  MoveL 5993 to (239.92, 153.82, 88.06) mm, rotated rx 180 ry 0 rz -180 deg; joints [-146.88, -81.725, -27.685, 63.006, 37.821, -57.184]
  MoveL 5994 to (239.92, 153.82, 88.06) mm, rotated rx 180 ry 0 rz -180 deg; joints [-146.88, -81.725, -27.685, 63.006, 37.821, -57.184]
  Call Extruder(262.09688)
  MoveL 5995 to (239.85, 154.05, 88.06) mm, rotated rx 180 ry 0 rz 180 deg; joints [-146.86, -81.738, -27.658, 63.04, 37.832, -57.218]
  MoveL 5996 to (239.85, 154.05, 88.06) mm, rotated rx 180 ry 0 rz 180 deg; joints [-146.86, -81.738, -27.658, 63.04, 37.832, -57.218]
  Call Extruder(262.22767)
  MoveL 5997 to (239.78, 154.27, 88.06) mm, rotated rx 180 ry 0 rz -180 deg; joints [-146.84, -81.752, -27.63, 63.073, 37.842, -57.252]
  MoveL 5998 to (239.78, 154.27, 88.06) mm, rotated rx 180 ry 0 rz -180 deg; joints [-146.84, -81.752, -27.63, 63.073, 37.842, -57.252]
  Call Extruder(262.35903)
  MoveL 5999 to (239.71, 154.49, 88.06) mm, rotated rx -180 ry 0 rz 180 deg; joints [-146.82, -81.765, -27.603, 63.107, 37.853, -57.286]
  MoveL 6000 to (239.71, 154.49, 88.06) mm, rotated rx -180 ry 0 rz 180 deg; joints [-146.82, -81.765, -27.603, 63.107, 37.853, -57.286]
  Call Extruder(262.47093)
  MoveL 6001 to (239.65, 154.68, 88.06) mm, rotated rx 180 ry 0 rz 180 deg; joints [-146.803, -81.776, -27.581, 63.135, 37.862, -57.314]
  MoveL 6002 to (239.65, 154.68, 88.06) mm, rotated rx 180 ry 0 rz 180 deg; joints [-146.803, -81.776, -27.581, 63.135, 37.862, -57.314]
  Call Extruder(262.58328)
  MoveL 6003 to (239.59, 154.87, 88.06) mm, rotated rx 180 ry 0 rz 180 deg; joints [-146.785, -81.787, -27.559, 63.163, 37.872, -57.342]
  MoveL 6004 to (239.59, 154.87, 88.06) mm, rotated rx 180 ry 0 rz 180 deg; joints [-146.785, -81.787, -27.559, 63.163, 37.872, -57.342]
  Call Extruder(262.69607)
  MoveL 6005 to (239.53, 155.06, 88.06) mm, rotated rx 180 ry 0 rz 180 deg; joints [-146.768, -81.798, -27.537, 63.19, 37.881, -57.37]
  MoveL 6006 to (239.53, 155.06, 88.06) mm, rotated rx 180 ry 0 rz 180 deg; joints [-146.768, -81.798, -27.537, 63.19, 37.881, -57.37]
  Call Extruder(262.80930)
  MoveL 6007 to (239.47, 155.25, 88.06) mm, rotated rx 180 ry 0 rz 180 deg; joints [-146.751, -81.808, -27.515, 63.218, 37.891, -57.398]
  MoveL 6008 to (239.47, 155.25, 88.06) mm, rotated rx 180 ry 0 rz 180 deg; joints [-146.751, -81.808, -27.515, 63.218, 37.891, -57.398]
  Call Extruder(262.92298)
  MoveL 6009 to (239.41, 155.44, 88.06) mm, rotated rx 180 ry 0 rz 180 deg; joints [-146.734, -81.819, -27.494, 63.246, 37.9, -57.426]
  MoveL 6010 to (239.41, 155.44, 88.06) mm, rotated rx 180 ry 0 rz 180 deg; joints [-146.734, -81.819, -27.494, 63.246, 37.9, -57.426]
  Call Extruder(263.10494)
  MoveL 6011 to (239.29, 155.73, 88.06) mm, rotated rx 180 ry 0 rz -180 deg; joints [-146.706, -81.832, -27.469, 63.285, 37.918, -57.464]
  MoveL 6012 to (239.29, 155.73, 88.06) mm, rotated rx 180 ry 0 rz -180 deg; joints [-146.706, -81.832, -27.469, 63.285, 37.918, -57.464]
  Call Extruder(263.28765)
  MoveL 6013 to (239.17, 156.02, 88.06) mm, rotated rx 180 ry 0 rz -180 deg; joints [-146.678, -81.844, -27.444, 63.323, 37.936, -57.501]
  MoveL 6014 to (239.17, 156.02, 88.06) mm, rotated rx 180 ry 0 rz -180 deg; joints [-146.678, -81.844, -27.444, 63.323, 37.936, -57.501]
  Call Extruder(263.45808)
  MoveL 6015 to (239.05, 156.29, 88.06) mm, rotated rx -180 ry 0 rz 180 deg; joints [-146.652, -81.855, -27.421, 63.359, 37.953, -57.535]
  MoveL 6016 to (239.05, 156.29, 88.06) mm, rotated rx -180 ry 0 rz 180 deg; joints [-146.652, -81.855, -27.421, 63.359, 37.953, -57.535]
  Call Extruder(263.61609)
  MoveL 6017 to (238.94, 156.54, 88.06) mm, rotated rx 180 ry 0 rz 180 deg; joints [-146.628, -81.865, -27.401, 63.392, 37.968, -57.567]
  MoveL 6018 to (238.94, 156.54, 88.06) mm, rotated rx 180 ry 0 rz 180 deg; joints [-146.628, -81.865, -27.401, 63.392, 37.968, -57.567]
  Call Extruder(263.77470)
  MoveL 6019 to (238.84, 156.79, 88.06) mm, rotated rx 180 ry 0 rz 180 deg; joints [-146.604, -81.875, -27.381, 63.424, 37.984, -57.598]
  MoveL 6020 to (238.84, 156.79, 88.06) mm, rotated rx 180 ry 0 rz 180 deg; joints [-146.604, -81.875, -27.381, 63.424, 37.984, -57.598]
  Call Extruder(263.98087)
  MoveL 6021 to (238.66, 157.09, 88.06) mm, rotated rx 180 ry 0 rz 180 deg; joints [-146.573, -81.879, -27.372, 63.457, 38.008, -57.626]
  MoveL 6022 to (238.66, 157.09, 88.06) mm, rotated rx 180 ry 0 rz 180 deg; joints [-146.573, -81.879, -27.372, 63.457, 38.008, -57.626]
  Call Extruder(264.18782)
  MoveL 6023 to (238.49, 157.4, 88.06) mm, rotated rx 180 ry 0 rz 180 deg; joints [-146.542, -81.883, -27.363, 63.489, 38.033, -57.654]
  MoveL 6024 to (238.49, 157.4, 88.06) mm, rotated rx 180 ry 0 rz 180 deg; joints [-146.542, -81.883, -27.363, 63.489, 38.033, -57.654]
  Call Extruder(264.39555)
  MoveL 6025 to (238.31, 157.7, 88.06) mm, rotated rx -180 ry 0 rz -180 deg; joints [-146.51, -81.888, -27.354, 63.522, 38.058, -57.682]
  MoveL 6026 to (238.31, 157.7, 88.06) mm, rotated rx -180 ry 0 rz -180 deg; joints [-146.51, -81.888, -27.354, 63.522, 38.058, -57.682]
  Call Extruder(264.60405)
  MoveL 6027 to (238.13, 158.01, 88.06) mm, rotated rx -180 ry 0 rz -180 deg; joints [-146.479, -81.892, -27.345, 63.554, 38.082, -57.71]
  MoveL 6028 to (238.13, 158.01, 88.06) mm, rotated rx -180 ry 0 rz -180 deg; joints [-146.479, -81.892, -27.345, 63.554, 38.082, -57.71]
  Call Extruder(264.78359)
  MoveL 6029 to (237.96, 158.25, 88.06) mm, rotated rx -180 ry 0 rz 180 deg; joints [-146.452, -81.89, -27.35, 63.575, 38.106, -57.725]
  MoveL 6030 to (237.96, 158.25, 88.06) mm, rotated rx -180 ry 0 rz 180 deg; joints [-146.452, -81.89, -27.35, 63.575, 38.106, -57.725]
  Call Extruder(265.11700)
  MoveL 6031 to (237.63, 158.7, 88.06) mm, rotated rx 180 ry 0 rz -180 deg; joints [-146.402, -81.885, -27.36, 63.612, 38.151, -57.752]
  MoveL 6032 to (237.63, 158.7, 88.06) mm, rotated rx 180 ry 0 rz -180 deg; joints [-146.402, -81.885, -27.36, 63.612, 38.151, -57.752]
  Call Extruder(265.45159)
  MoveL 6033 to (237.3, 159.15, 88.06) mm, rotated rx -180 ry 0 rz 180 deg; joints [-146.352, -81.88, -27.37, 63.65, 38.195, -57.779]
  Call Extruder(266.27956)
  MoveL 6034 to (236.39, 160.19, 88.06) mm, rotated rx 180 ry 0 rz 180 deg; joints [-146.229, -81.842, -27.447, 63.711, 38.316, -57.805]
  Call Extruder(267.10747)
  MoveL 6035 to (235.35, 161.1, 88.06) mm, rotated rx -180 ry 0 rz 180 deg; joints [-146.109, -81.769, -27.595, 63.729, 38.451, -57.777]
  Call Extruder(267.27478)
  MoveL 6036 to (235.13, 161.27, 88.06) mm, rotated rx -180 ry 0 rz 180 deg; joints [-146.086, -81.749, -27.636, 63.726, 38.48, -57.764]
  MoveL 6037 to (235.13, 161.27, 88.06) mm, rotated rx -180 ry 0 rz 180 deg; joints [-146.086, -81.749, -27.636, 63.726, 38.48, -57.764]
  Call Extruder(267.60821)
  MoveL 6038 to (234.68, 161.59, 88.06) mm, rotated rx 180 ry 0 rz 180 deg; joints [-146.039, -81.71, -27.716, 63.721, 38.537, -57.737]
  MoveL 6039 to (234.68, 161.59, 88.06) mm, rotated rx 180 ry 0 rz 180 deg; joints [-146.039, -81.71, -27.716, 63.721, 38.537, -57.737]
  Call Extruder(267.94046)
  MoveL 6040 to (234.23, 161.92, 88.06) mm, rotated rx -180 ry 0 rz 180 deg; joints [-145.992, -81.67, -27.795, 63.716, 38.595, -57.71]
  MoveL 6041 to (234.23, 161.92, 88.06) mm, rotated rx -180 ry 0 rz 180 deg; joints [-145.992, -81.67, -27.795, 63.716, 38.595, -57.71]
  Call Extruder(268.05811)
  MoveL 6042 to (234.05, 162.02, 88.06) mm, rotated rx -180 ry 0 rz -180 deg; joints [-145.976, -81.653, -27.831, 63.709, 38.617, -57.695]
  MoveL 6043 to (234.05, 162.02, 88.06) mm, rotated rx -180 ry 0 rz -180 deg; joints [-145.976, -81.653, -27.831, 63.709, 38.617, -57.695]
  Call Extruder(268.26584)
  MoveL 6044 to (233.75, 162.2, 88.06) mm, rotated rx -180 ry 0 rz 180 deg; joints [-145.947, -81.621, -27.895, 63.697, 38.655, -57.667]
  MoveL 6045 to (233.75, 162.2, 88.06) mm, rotated rx -180 ry 0 rz 180 deg; joints [-145.947, -81.621, -27.895, 63.697, 38.655, -57.667]
  Call Extruder(268.47279)
  MoveL 6046 to (233.45, 162.37, 88.06) mm, rotated rx -180 ry 0 rz 180 deg; joints [-145.919, -81.59, -27.959, 63.685, 38.693, -57.64]
  MoveL 6047 to (233.45, 162.37, 88.06) mm, rotated rx -180 ry 0 rz 180 deg; joints [-145.919, -81.59, -27.959, 63.685, 38.693, -57.64]
  Call Extruder(268.67896)
  MoveL 6048 to (233.14, 162.55, 88.06) mm, rotated rx 180 ry 0 rz 180 deg; joints [-145.891, -81.558, -28.023, 63.673, 38.732, -57.613]
  MoveL 6049 to (233.14, 162.55, 88.06) mm, rotated rx 180 ry 0 rz 180 deg; joints [-145.891, -81.558, -28.023, 63.673, 38.732, -57.613]
  Call Extruder(268.86063)
  MoveL 6050 to (232.87, 162.69, 88.06) mm, rotated rx 180 ry 0 rz 180 deg; joints [-145.866, -81.528, -28.085, 63.659, 38.766, -57.584]
  MoveL 6051 to (232.87, 162.69, 88.06) mm, rotated rx 180 ry 0 rz 180 deg; joints [-145.866, -81.528, -28.085, 63.659, 38.766, -57.584]
  Call Extruder(269.01860)
  MoveL 6052 to (232.62, 162.8, 88.06) mm, rotated rx -180 ry 0 rz -180 deg; joints [-145.845, -81.498, -28.145, 63.642, 38.797, -57.554]
  MoveL 6053 to (232.62, 162.8, 88.06) mm, rotated rx -180 ry 0 rz -180 deg; joints [-145.845, -81.498, -28.145, 63.642, 38.797, -57.554]
  Call Extruder(269.17597)
  MoveL 6054 to (232.37, 162.9, 88.06) mm, rotated rx -180 ry 0 rz 180 deg; joints [-145.825, -81.468, -28.205, 63.626, 38.828, -57.524]
  MoveL 6055 to (232.37, 162.9, 88.06) mm, rotated rx -180 ry 0 rz 180 deg; joints [-145.825, -81.468, -28.205, 63.626, 38.828, -57.524]
  Call Extruder(269.35871)
  MoveL 6056 to (232.07, 163.03, 88.06) mm, rotated rx -180 ry 0 rz 180 deg; joints [-145.801, -81.433, -28.277, 63.606, 38.864, -57.488]
  MoveL 6057 to (232.07, 163.03, 88.06) mm, rotated rx -180 ry 0 rz 180 deg; joints [-145.801, -81.433, -28.277, 63.606, 38.864, -57.488]
  Call Extruder(269.54070)
  MoveL 6058 to (231.78, 163.15, 88.06) mm, rotated rx -180 ry 0 rz -180 deg; joints [-145.777, -81.397, -28.349, 63.586, 38.9, -57.452]
  MoveL 6059 to (231.78, 163.15, 88.06) mm, rotated rx -180 ry 0 rz -180 deg; joints [-145.777, -81.397, -28.349, 63.586, 38.9, -57.452]
  Call Extruder(269.68804)
  MoveL 6060 to (231.54, 163.24, 88.06) mm, rotated rx -180 ry 0 rz -180 deg; joints [-145.759, -81.368, -28.409, 63.568, 38.93, -57.421]
  MoveL 6061 to (231.54, 163.24, 88.06) mm, rotated rx -180 ry 0 rz -180 deg; joints [-145.759, -81.368, -28.409, 63.568, 38.93, -57.421]
  Call Extruder(269.80126)
  MoveL 6062 to (231.35, 163.3, 88.06) mm, rotated rx 180 ry 0 rz 180 deg; joints [-145.744, -81.343, -28.459, 63.552, 38.953, -57.394]
  MoveL 6063 to (231.35, 163.3, 88.06) mm, rotated rx 180 ry 0 rz 180 deg; joints [-145.744, -81.343, -28.459, 63.552, 38.953, -57.394]
  Call Extruder(269.91404)
  MoveL 6064 to (231.17, 163.36, 88.06) mm, rotated rx -180 ry 0 rz 180 deg; joints [-145.73, -81.319, -28.509, 63.536, 38.976, -57.368]
  MoveL 6065 to (231.17, 163.36, 88.06) mm, rotated rx -180 ry 0 rz 180 deg; joints [-145.73, -81.319, -28.509, 63.536, 38.976, -57.368]
  Call Extruder(270.02637)
  MoveL 6066 to (230.98, 163.42, 88.06) mm, rotated rx 180 ry 0 rz 180 deg; joints [-145.716, -81.294, -28.559, 63.52, 38.999, -57.341]
  MoveL 6067 to (230.98, 163.42, 88.06) mm, rotated rx 180 ry 0 rz 180 deg; joints [-145.716, -81.294, -28.559, 63.52, 38.999, -57.341]
  Call Extruder(270.13826)
  MoveL 6068 to (230.79, 163.48, 88.06) mm, rotated rx 180 ry 0 rz -180 deg; joints [-145.702, -81.27, -28.608, 63.505, 39.022, -57.315]
  MoveL 6069 to (230.79, 163.48, 88.06) mm, rotated rx 180 ry 0 rz -180 deg; joints [-145.702, -81.27, -28.608, 63.505, 39.022, -57.315]
  Call Extruder(270.25966)
  MoveL 6070 to (230.58, 163.55, 88.06) mm, rotated rx 180 ry 0 rz 180 deg; joints [-145.687, -81.243, -28.663, 63.487, 39.048, -57.286]
  MoveL 6071 to (230.58, 163.55, 88.06) mm, rotated rx 180 ry 0 rz 180 deg; joints [-145.687, -81.243, -28.663, 63.487, 39.048, -57.286]
  Call Extruder(270.39048)
  MoveL 6072 to (230.36, 163.61, 88.06) mm, rotated rx -180 ry 0 rz 180 deg; joints [-145.67, -81.213, -28.722, 63.468, 39.075, -57.253]
  MoveL 6073 to (230.36, 163.61, 88.06) mm, rotated rx -180 ry 0 rz 180 deg; joints [-145.67, -81.213, -28.722, 63.468, 39.075, -57.253]
  Call Extruder(270.52072)
  MoveL 6074 to (230.14, 163.68, 88.06) mm, rotated rx 180 ry 0 rz 180 deg; joints [-145.654, -81.184, -28.782, 63.449, 39.102, -57.221]
  MoveL 6075 to (230.14, 163.68, 88.06) mm, rotated rx 180 ry 0 rz 180 deg; joints [-145.654, -81.184, -28.782, 63.449, 39.102, -57.221]
  Call Extruder(270.65041)
  MoveL 6076 to (229.91, 163.75, 88.06) mm, rotated rx 180 ry 0 rz 180 deg; joints [-145.638, -81.154, -28.842, 63.429, 39.13, -57.189]
  MoveL 6077 to (229.91, 163.75, 88.06) mm, rotated rx 180 ry 0 rz 180 deg; joints [-145.638, -81.154, -28.842, 63.429, 39.13, -57.189]
  Call Extruder(270.77952)
  MoveL 6078 to (229.69, 163.82, 88.06) mm, rotated rx -180 ry 0 rz 180 deg; joints [-145.621, -81.125, -28.902, 63.41, 39.157, -57.157]
  MoveL 6079 to (229.69, 163.82, 88.06) mm, rotated rx -180 ry 0 rz 180 deg; joints [-145.621, -81.125, -28.902, 63.41, 39.157, -57.157]
  Call Extruder(270.89460)
  MoveL 6080 to (229.48, 163.86, 88.06) mm, rotated rx -180 ry 0 rz 180 deg; joints [-145.607, -81.096, -28.96, 63.39, 39.182, -57.125]
  MoveL 6081 to (229.48, 163.86, 88.06) mm, rotated rx -180 ry 0 rz 180 deg; joints [-145.607, -81.096, -28.96, 63.39, 39.182, -57.125]
  Call Extruder(271.00922)
  MoveL 6082 to (229.28, 163.91, 88.06) mm, rotated rx 180 ry 0 rz -180 deg; joints [-145.594, -81.068, -29.017, 63.369, 39.206, -57.092]
  MoveL 6083 to (229.28, 163.91, 88.06) mm, rotated rx 180 ry 0 rz -180 deg; joints [-145.594, -81.068, -29.017, 63.369, 39.206, -57.092]
  Call Extruder(271.12339)
  MoveL 6084 to (229.08, 163.95, 88.06) mm, rotated rx -180 ry 0 rz 180 deg; joints [-145.58, -81.039, -29.076, 63.349, 39.231, -57.06]
  MoveL 6085 to (229.08, 163.95, 88.06) mm, rotated rx -180 ry 0 rz 180 deg; joints [-145.58, -81.039, -29.076, 63.349, 39.231, -57.06]
  Call Extruder(271.23711)
  MoveL 6086 to (228.87, 164, 88.06) mm, rotated rx -180 ry 0 rz 180 deg; joints [-145.566, -81.011, -29.134, 63.328, 39.256, -57.027]
  MoveL 6087 to (228.87, 164, 88.06) mm, rotated rx -180 ry 0 rz 180 deg; joints [-145.566, -81.011, -29.134, 63.328, 39.256, -57.027]
  Call Extruder(271.36253)
  MoveL 6088 to (228.65, 164.04, 88.06) mm, rotated rx 180 ry 0 rz 180 deg; joints [-145.551, -80.979, -29.198, 63.305, 39.283, -56.991]
  MoveL 6089 to (228.65, 164.04, 88.06) mm, rotated rx 180 ry 0 rz 180 deg; joints [-145.551, -80.979, -29.198, 63.305, 39.283, -56.991]
  Call Extruder(271.49950)
  MoveL 6090 to (228.4, 164.09, 88.06) mm, rotated rx -180 ry 0 rz 180 deg; joints [-145.535, -80.944, -29.269, 63.28, 39.313, -56.951]
  MoveL 6091 to (228.4, 164.09, 88.06) mm, rotated rx -180 ry 0 rz 180 deg; joints [-145.535, -80.944, -29.269, 63.28, 39.313, -56.951]
  Call Extruder(271.63587)
  MoveL 6092 to (228.15, 164.14, 88.06) mm, rotated rx -180 ry 0 rz 180 deg; joints [-145.518, -80.909, -29.341, 63.254, 39.344, -56.91]
  MoveL 6093 to (228.15, 164.14, 88.06) mm, rotated rx -180 ry 0 rz 180 deg; joints [-145.518, -80.909, -29.341, 63.254, 39.344, -56.91]
  Call Extruder(271.77163)
  MoveL 6094 to (227.9, 164.19, 88.06) mm, rotated rx 180 ry 0 rz 180 deg; joints [-145.502, -80.874, -29.412, 63.229, 39.374, -56.87]
  MoveL 6095 to (227.9, 164.19, 88.06) mm, rotated rx 180 ry 0 rz 180 deg; joints [-145.502, -80.874, -29.412, 63.229, 39.374, -56.87]
  Call Extruder(271.90678)
  MoveL 6096 to (227.65, 164.24, 88.06) mm, rotated rx 180 ry 0 rz 180 deg; joints [-145.485, -80.839, -29.483, 63.204, 39.404, -56.831]
  MoveL 6097 to (227.65, 164.24, 88.06) mm, rotated rx 180 ry 0 rz 180 deg; joints [-145.485, -80.839, -29.483, 63.204, 39.404, -56.831]
  Call Extruder(272.04131)
  MoveL 6098 to (227.4, 164.29, 88.06) mm, rotated rx 180 ry 0 rz 180 deg; joints [-145.469, -80.804, -29.554, 63.179, 39.434, -56.791]
  MoveL 6099 to (227.4, 164.29, 88.06) mm, rotated rx 180 ry 0 rz 180 deg; joints [-145.469, -80.804, -29.554, 63.179, 39.434, -56.791]
  Call Extruder(272.17524)
  MoveL 6100 to (227.15, 164.34, 88.06) mm, rotated rx 180 ry 0 rz -180 deg; joints [-145.453, -80.769, -29.625, 63.154, 39.464, -56.751]
  MoveL 6101 to (227.15, 164.34, 88.06) mm, rotated rx 180 ry 0 rz -180 deg; joints [-145.453, -80.769, -29.625, 63.154, 39.464, -56.751]
  Call Extruder(272.32310)
  MoveL 6102 to (226.87, 164.39, 88.06) mm, rotated rx 180 ry 0 rz -180 deg; joints [-145.435, -80.73, -29.705, 63.126, 39.497, -56.706]
  MoveL 6103 to (226.87, 164.39, 88.06) mm, rotated rx 180 ry 0 rz -180 deg; joints [-145.435, -80.73, -29.705, 63.126, 39.497, -56.706]
  Call Extruder(272.48484)
  MoveL 6104 to (226.57, 164.44, 88.06) mm, rotated rx 180 ry 0 rz -180 deg; joints [-145.415, -80.686, -29.794, 63.093, 39.534, -56.655]
  MoveL 6105 to (226.57, 164.44, 88.06) mm, rotated rx 180 ry 0 rz -180 deg; joints [-145.415, -80.686, -29.794, 63.093, 39.534, -56.655]
  Call Extruder(272.64586)
  MoveL 6106 to (226.26, 164.49, 88.06) mm, rotated rx -180 ry 0 rz -180 deg; joints [-145.396, -80.642, -29.884, 63.061, 39.57, -56.605]
  MoveL 6107 to (226.26, 164.49, 88.06) mm, rotated rx -180 ry 0 rz -180 deg; joints [-145.396, -80.642, -29.884, 63.061, 39.57, -56.605]
  Call Extruder(272.80614)
  MoveL 6108 to (225.96, 164.54, 88.06) mm, rotated rx 180 ry 0 rz 180 deg; joints [-145.377, -80.598, -29.973, 63.029, 39.607, -56.554]
  MoveL 6109 to (225.96, 164.54, 88.06) mm, rotated rx 180 ry 0 rz 180 deg; joints [-145.377, -80.598, -29.973, 63.029, 39.607, -56.554]
  Call Extruder(272.96570)
  MoveL 6110 to (225.65, 164.58, 88.06) mm, rotated rx 180 ry 0 rz -180 deg; joints [-145.357, -80.555, -30.061, 62.997, 39.644, -56.504]
  MoveL 6111 to (225.65, 164.58, 88.06) mm, rotated rx 180 ry 0 rz -180 deg; joints [-145.357, -80.555, -30.061, 62.997, 39.644, -56.504]
  Call Extruder(273.12452)
  MoveL 6112 to (225.34, 164.63, 88.06) mm, rotated rx 180 ry 0 rz 180 deg; joints [-145.338, -80.511, -30.15, 62.965, 39.68, -56.454]
  MoveL 6113 to (225.34, 164.63, 88.06) mm, rotated rx 180 ry 0 rz 180 deg; joints [-145.338, -80.511, -30.15, 62.965, 39.68, -56.454]
  Call Extruder(273.30319)
  MoveL 6114 to (225, 164.68, 88.06) mm, rotated rx -180 ry 0 rz 180 deg; joints [-145.317, -80.461, -30.252, 62.928, 39.722, -56.396]
  MoveL 6115 to (225, 164.68, 88.06) mm, rotated rx -180 ry 0 rz 180 deg; joints [-145.317, -80.461, -30.252, 62.928, 39.722, -56.396]
  Call Extruder(273.50164)
  MoveL 6116 to (224.61, 164.72, 88.06) mm, rotated rx -180 ry 0 rz -180 deg; joints [-145.293, -80.405, -30.366, 62.886, 39.768, -56.33]
  MoveL 6117 to (224.61, 164.72, 88.06) mm, rotated rx -180 ry 0 rz -180 deg; joints [-145.293, -80.405, -30.366, 62.886, 39.768, -56.33]
  Call Extruder(273.69921)
  MoveL 6118 to (224.22, 164.77, 88.06) mm, rotated rx -180 ry 0 rz 180 deg; joints [-145.27, -80.349, -30.481, 62.844, 39.814, -56.265]
  MoveL 6119 to (224.22, 164.77, 88.06) mm, rotated rx -180 ry 0 rz 180 deg; joints [-145.27, -80.349, -30.481, 62.844, 39.814, -56.265]
  Call Extruder(273.89592)
  MoveL 6120 to (223.84, 164.82, 88.06) mm, rotated rx -180 ry 0 rz 180 deg; joints [-145.246, -80.293, -30.595, 62.802, 39.86, -56.199]
  MoveL 6121 to (223.84, 164.82, 88.06) mm, rotated rx -180 ry 0 rz 180 deg; joints [-145.246, -80.293, -30.595, 62.802, 39.86, -56.199]
  Call Extruder(274.09176)
  MoveL 6122 to (223.45, 164.86, 88.06) mm, rotated rx -180 ry 0 rz 180 deg; joints [-145.223, -80.237, -30.71, 62.76, 39.906, -56.134]
  MoveL 6123 to (223.45, 164.86, 88.06) mm, rotated rx -180 ry 0 rz 180 deg; joints [-145.223, -80.237, -30.71, 62.76, 39.906, -56.134]
  Call Extruder(274.38712)
  MoveL 6124 to (222.86, 164.91, 88.06) mm, rotated rx 180 ry 0 rz 180 deg; joints [-145.189, -80.149, -30.888, 62.694, 39.976, -56.031]
  MoveL 6125 to (222.86, 164.91, 88.06) mm, rotated rx 180 ry 0 rz 180 deg; joints [-145.189, -80.149, -30.888, 62.694, 39.976, -56.031]
  Call Extruder(274.68114)
  MoveL 6126 to (222.27, 164.96, 88.06) mm, rotated rx 180 ry 0 rz 180 deg; joints [-145.155, -80.063, -31.065, 62.628, 40.046, -55.929]
  MoveL 6127 to (222.27, 164.96, 88.06) mm, rotated rx 180 ry 0 rz 180 deg; joints [-145.155, -80.063, -31.065, 62.628, 40.046, -55.929]
  Call Extruder(274.97384)
  MoveL 6128 to (221.68, 165, 88.06) mm, rotated rx 180 ry 0 rz 180 deg; joints [-145.121, -79.976, -31.241, 62.563, 40.115, -55.828]
  MoveL 6129 to (221.68, 165, 88.06) mm, rotated rx 180 ry 0 rz 180 deg; joints [-145.121, -79.976, -31.241, 62.563, 40.115, -55.828]
  Call Extruder(275.54729)
  MoveL 6130 to (220.52, 165.05, 88.06) mm, rotated rx 180 ry 0 rz -180 deg; joints [-145.056, -79.802, -31.597, 62.428, 40.252, -55.621]
  MoveL 6131 to (220.52, 165.05, 88.06) mm, rotated rx 180 ry 0 rz -180 deg; joints [-145.056, -79.802, -31.597, 62.428, 40.252, -55.621]
  Call Extruder(276.26129)
  MoveL 6132 to (219.06, 165.09, 88.06) mm, rotated rx 180 ry 0 rz -180 deg; joints [-144.977, -79.585, -32.042, 62.26, 40.423, -55.363]
  Call Extruder(393.10803)
  MoveL 6133 to (-19.06, 165.09, 88.06) mm, rotated rx -180 ry 0 rz 180 deg; joints [-127.435, -59.057, -77.147, 61.077, 65.122, -37.284]
  Call Extruder(393.53664)
  MoveL 6134 to (-19.94, 165.07, 88.06) mm, rotated rx 180 ry 0 rz 180 deg; joints [-127.348, -59.012, -77.256, 61.127, 65.205, -37.254]
  MoveL 6135 to (-19.94, 165.07, 88.06) mm, rotated rx 180 ry 0 rz 180 deg; joints [-127.348, -59.012, -77.256, 61.127, 65.205, -37.254]
  Call Extruder(394.11009)
  MoveL 6136 to (-21.1, 165.03, 88.06) mm, rotated rx 180 ry 0 rz 180 deg; joints [-127.235, -58.952, -77.404, 61.191, 65.316, -37.211]
  MoveL 6137 to (-21.1, 165.03, 88.06) mm, rotated rx 180 ry 0 rz 180 deg; joints [-127.235, -58.952, -77.404, 61.191, 65.316, -37.211]
  Call Extruder(394.54439)
  MoveL 6138 to (-21.97, 164.98, 88.06) mm, rotated rx 180 ry 0 rz -180 deg; joints [-127.15, -58.906, -77.517, 61.238, 65.4, -37.178]
  MoveL 6139 to (-21.97, 164.98, 88.06) mm, rotated rx 180 ry 0 rz -180 deg; joints [-127.15, -58.906, -77.517, 61.238, 65.4, -37.178]
  Call Extruder(394.83842)
  MoveL 6140 to (-22.56, 164.93, 88.06) mm, rotated rx -180 ry 0 rz 180 deg; joints [-127.093, -58.875, -77.595, 61.269, 65.456, -37.153]
  MoveL 6141 to (-22.56, 164.93, 88.06) mm, rotated rx -180 ry 0 rz 180 deg; joints [-127.093, -58.875, -77.595, 61.269, 65.456, -37.153]
  Call Extruder(395.13378)
  MoveL 6142 to (-23.15, 164.89, 88.06) mm, rotated rx -180 ry 0 rz -180 deg; joints [-127.037, -58.843, -77.673, 61.3, 65.512, -37.129]
  MoveL 6143 to (-23.15, 164.89, 88.06) mm, rotated rx -180 ry 0 rz -180 deg; joints [-127.037, -58.843, -77.673, 61.3, 65.512, -37.129]
  Call Extruder(395.37999)
  MoveL 6144 to (-23.64, 164.84, 88.06) mm, rotated rx 180 ry 0 rz -180 deg; joints [-126.991, -58.816, -77.739, 61.324, 65.559, -37.108]
  MoveL 6145 to (-23.64, 164.84, 88.06) mm, rotated rx 180 ry 0 rz -180 deg; joints [-126.991, -58.816, -77.739, 61.324, 65.559, -37.108]
  Call Extruder(395.57670)
  MoveL 6146 to (-24.03, 164.79, 88.06) mm, rotated rx 180 ry 0 rz -180 deg; joints [-126.955, -58.794, -77.792, 61.343, 65.596, -37.09]
  MoveL 6147 to (-24.03, 164.79, 88.06) mm, rotated rx 180 ry 0 rz -180 deg; joints [-126.955, -58.794, -77.792, 61.343, 65.596, -37.09]
  Call Extruder(395.77427)
  MoveL 6148 to (-24.42, 164.75, 88.06) mm, rotated rx 180 ry 0 rz 180 deg; joints [-126.919, -58.773, -77.846, 61.362, 65.633, -37.073]
  MoveL 6149 to (-24.42, 164.75, 88.06) mm, rotated rx 180 ry 0 rz 180 deg; joints [-126.919, -58.773, -77.846, 61.362, 65.633, -37.073]
  Call Extruder(395.97271)
  MoveL 6150 to (-24.8, 164.7, 88.06) mm, rotated rx 180 ry 0 rz 180 deg; joints [-126.883, -58.751, -77.899, 61.381, 65.67, -37.055]
  MoveL 6151 to (-24.8, 164.7, 88.06) mm, rotated rx 180 ry 0 rz 180 deg; joints [-126.883, -58.751, -77.899, 61.381, 65.67, -37.055]
  Call Extruder(396.17202)
  MoveL 6152 to (-25.19, 164.66, 88.06) mm, rotated rx -180 ry 0 rz 180 deg; joints [-126.847, -58.729, -77.953, 61.4, 65.706, -37.037]
  MoveL 6153 to (-25.19, 164.66, 88.06) mm, rotated rx -180 ry 0 rz 180 deg; joints [-126.847, -58.729, -77.953, 61.4, 65.706, -37.037]
  Call Extruder(396.33085)
  MoveL 6154 to (-25.5, 164.61, 88.06) mm, rotated rx 180 ry 0 rz 180 deg; joints [-126.82, -58.712, -77.997, 61.414, 65.736, -37.022]
  MoveL 6155 to (-25.5, 164.61, 88.06) mm, rotated rx 180 ry 0 rz 180 deg; joints [-126.82, -58.712, -77.997, 61.414, 65.736, -37.022]
  Call Extruder(396.49041)
  MoveL 6156 to (-25.8, 164.56, 88.06) mm, rotated rx -180 ry 0 rz 180 deg; joints [-126.792, -58.694, -78.041, 61.427, 65.765, -37.007]
  MoveL 6157 to (-25.8, 164.56, 88.06) mm, rotated rx -180 ry 0 rz 180 deg; joints [-126.792, -58.694, -78.041, 61.427, 65.765, -37.007]
  Call Extruder(396.65070)
  MoveL 6158 to (-26.11, 164.51, 88.06) mm, rotated rx 180 ry 0 rz -180 deg; joints [-126.765, -58.676, -78.085, 61.441, 65.794, -36.991]
  MoveL 6159 to (-26.11, 164.51, 88.06) mm, rotated rx 180 ry 0 rz -180 deg; joints [-126.765, -58.676, -78.085, 61.441, 65.794, -36.991]
  Call Extruder(396.81172)
  MoveL 6160 to (-26.41, 164.46, 88.06) mm, rotated rx 180 ry 0 rz 180 deg; joints [-126.737, -58.658, -78.129, 61.455, 65.823, -36.976]
  MoveL 6161 to (-26.41, 164.46, 88.06) mm, rotated rx 180 ry 0 rz 180 deg; joints [-126.737, -58.658, -78.129, 61.455, 65.823, -36.976]
  Call Extruder(396.97346)
  MoveL 6162 to (-26.72, 164.41, 88.06) mm, rotated rx 180 ry 0 rz -180 deg; joints [-126.71, -58.64, -78.173, 61.469, 65.852, -36.961]
  MoveL 6163 to (-26.72, 164.41, 88.06) mm, rotated rx 180 ry 0 rz -180 deg; joints [-126.71, -58.64, -78.173, 61.469, 65.852, -36.961]
  Call Extruder(397.13593)
  MoveL 6164 to (-27.03, 164.36, 88.06) mm, rotated rx -180 ry 0 rz -180 deg; joints [-126.682, -58.623, -78.216, 61.483, 65.881, -36.945]
  MoveL 6165 to (-27.03, 164.36, 88.06) mm, rotated rx -180 ry 0 rz -180 deg; joints [-126.682, -58.623, -78.216, 61.483, 65.881, -36.945]
  Call Extruder(397.26986)
  MoveL 6166 to (-27.27, 164.32, 88.06) mm, rotated rx -180 ry 0 rz -180 deg; joints [-126.66, -58.608, -78.254, 61.493, 65.905, -36.932]
  MoveL 6167 to (-27.27, 164.32, 88.06) mm, rotated rx -180 ry 0 rz -180 deg; joints [-126.66, -58.608, -78.254, 61.493, 65.905, -36.932]
  Call Extruder(397.40439)
  MoveL 6168 to (-27.52, 164.27, 88.06) mm, rotated rx 180 ry 0 rz 180 deg; joints [-126.638, -58.593, -78.291, 61.503, 65.928, -36.918]
  MoveL 6169 to (-27.52, 164.27, 88.06) mm, rotated rx 180 ry 0 rz 180 deg; joints [-126.638, -58.593, -78.291, 61.503, 65.928, -36.918]
  Call Extruder(397.53954)
  MoveL 6170 to (-27.77, 164.22, 88.06) mm, rotated rx -180 ry 0 rz 180 deg; joints [-126.617, -58.577, -78.328, 61.514, 65.952, -36.905]
  MoveL 6171 to (-27.77, 164.22, 88.06) mm, rotated rx -180 ry 0 rz 180 deg; joints [-126.617, -58.577, -78.328, 61.514, 65.952, -36.905]
  Call Extruder(397.67530)
  MoveL 6172 to (-28.02, 164.17, 88.06) mm, rotated rx 180 ry 0 rz 180 deg; joints [-126.595, -58.563, -78.365, 61.524, 65.976, -36.891]
  MoveL 6173 to (-28.02, 164.17, 88.06) mm, rotated rx 180 ry 0 rz 180 deg; joints [-126.595, -58.563, -78.365, 61.524, 65.976, -36.891]
  Call Extruder(397.81166)
  MoveL 6174 to (-28.27, 164.12, 88.06) mm, rotated rx 180 ry 0 rz 180 deg; joints [-126.573, -58.547, -78.403, 61.534, 65.999, -36.878]
  MoveL 6175 to (-28.27, 164.12, 88.06) mm, rotated rx 180 ry 0 rz 180 deg; joints [-126.573, -58.547, -78.403, 61.534, 65.999, -36.878]
  Call Extruder(397.89653)
  MoveL 6176 to (-28.43, 164.09, 88.06) mm, rotated rx 180 ry 0 rz 180 deg; joints [-126.559, -58.538, -78.426, 61.541, 66.014, -36.869]
  Set speed (130.0 mm/s)
  MoveL 6177 to (-31.76, 163.31, 88.06) mm, rotated rx 180 ry 0 rz 180 deg; joints [-126.274, -58.332, -78.939, 61.672, 66.331, -36.675]
  MoveL 6178 to (-31.76, 163.31, 97.46) mm, rotated rx 180 ry 0 rz 180 deg; joints [-126.274, -57.059, -79.517, 61.942, 66.003, -37.344]
  Call Extruder(395.89653)
  Set speed (40.0 mm/s)
  MoveL 6179 to (-31.76, 163.31, 97.46) mm, rotated rx 180 ry 0 rz 180 deg; joints [-126.274, -57.059, -79.517, 61.942, 66.003, -37.344]
  Call Extruder(0.00000)
  Set speed (130.0 mm/s)
  MoveL 6180 to (-31.64, 163.21, 97.46) mm, rotated rx 180 ry 0 rz 180 deg; joints [-126.294, -57.059, -79.519, 61.924, 65.991, -37.336]
  Call Extruder(2.00000)
  Set speed (40.0 mm/s)
  MoveL 6181 to (-31.64, 163.21, 97.46) mm, rotated rx 180 ry 0 rz 180 deg; joints [-126.294, -57.059, -79.519, 61.924, 65.991, -37.336]
  Set speed (30.0 mm/s)
  MoveL 6182 to (-31.64, 163.21, 97.46) mm, rotated rx 180 ry 0 rz 180 deg; joints [-126.294, -57.059, -79.519, 61.924, 65.991, -37.336]
  Call Extruder(2.18198)
  MoveL 6183 to (-31.93, 163.09, 97.46) mm, rotated rx 180 ry 0 rz 180 deg; joints [-126.273, -57.037, -79.572, 61.93, 66.018, -37.313]
  MoveL 6184 to (-31.93, 163.09, 97.46) mm, rotated rx 180 ry 0 rz 180 deg; joints [-126.273, -57.037, -79.572, 61.93, 66.018, -37.313]
  Call Extruder(2.36471)
  MoveL 6185 to (-32.22, 162.96, 97.46) mm, rotated rx 180 ry 0 rz 180 deg; joints [-126.252, -57.015, -79.625, 61.936, 66.046, -37.291]
  MoveL 6186 to (-32.22, 162.96, 97.46) mm, rotated rx 180 ry 0 rz 180 deg; joints [-126.252, -57.015, -79.625, 61.936, 66.046, -37.291]
  Call Extruder(2.53513)
  MoveL 6187 to (-32.49, 162.85, 97.46) mm, rotated rx 180 ry 0 rz 180 deg; joints [-126.233, -56.995, -79.674, 61.942, 66.072, -37.269]
  MoveL 6188 to (-32.49, 162.85, 97.46) mm, rotated rx 180 ry 0 rz 180 deg; joints [-126.233, -56.995, -79.674, 61.942, 66.072, -37.269]
  Call Extruder(2.69310)
  MoveL 6189 to (-32.74, 162.74, 97.46) mm, rotated rx -180 ry 0 rz 180 deg; joints [-126.215, -56.976, -79.72, 61.947, 66.095, -37.249]
  MoveL 6190 to (-32.74, 162.74, 97.46) mm, rotated rx -180 ry 0 rz 180 deg; joints [-126.215, -56.976, -79.72, 61.947, 66.095, -37.249]
  Call Extruder(2.85168)
  MoveL 6191 to (-32.99, 162.64, 97.46) mm, rotated rx 180 ry 0 rz 180 deg; joints [-126.197, -56.957, -79.766, 61.952, 66.119, -37.23]
  MoveL 6192 to (-32.99, 162.64, 97.46) mm, rotated rx 180 ry 0 rz 180 deg; joints [-126.197, -56.957, -79.766, 61.952, 66.119, -37.23]
  Call Extruder(3.05785)
  MoveL 6193 to (-33.29, 162.46, 97.46) mm, rotated rx 180 ry 0 rz 180 deg; joints [-126.179, -56.932, -79.829, 61.953, 66.147, -37.2]
  MoveL 6194 to (-33.29, 162.46, 97.46) mm, rotated rx 180 ry 0 rz 180 deg; joints [-126.179, -56.932, -79.829, 61.953, 66.147, -37.2]
  Call Extruder(3.26479)
  MoveL 6195 to (-33.6, 162.29, 97.46) mm, rotated rx 180 ry 0 rz 180 deg; joints [-126.16, -56.906, -79.892, 61.955, 66.176, -37.171]
  MoveL 6196 to (-33.6, 162.29, 97.46) mm, rotated rx 180 ry 0 rz 180 deg; joints [-126.16, -56.906, -79.892, 61.955, 66.176, -37.171]
  Call Extruder(3.47251)
  MoveL 6197 to (-33.9, 162.11, 97.46) mm, rotated rx 180 ry 0 rz 180 deg; joints [-126.142, -56.88, -79.955, 61.956, 66.204, -37.141]
  MoveL 6198 to (-33.9, 162.11, 97.46) mm, rotated rx 180 ry 0 rz 180 deg; joints [-126.142, -56.88, -79.955, 61.956, 66.204, -37.141]
  Call Extruder(3.68101)
  MoveL 6199 to (-34.21, 161.93, 97.46) mm, rotated rx -180 ry 0 rz 180 deg; joints [-126.123, -56.854, -80.018, 61.958, 66.233, -37.112]
  MoveL 6200 to (-34.21, 161.93, 97.46) mm, rotated rx -180 ry 0 rz 180 deg; joints [-126.123, -56.854, -80.018, 61.958, 66.233, -37.112]
  Call Extruder(3.86055)
  MoveL 6201 to (-34.45, 161.76, 97.46) mm, rotated rx 180 ry 0 rz 180 deg; joints [-126.111, -56.831, -80.074, 61.955, 66.256, -37.084]
  MoveL 6202 to (-34.45, 161.76, 97.46) mm, rotated rx 180 ry 0 rz 180 deg; joints [-126.111, -56.831, -80.074, 61.955, 66.256, -37.084]
  Call Extruder(4.19399)
  MoveL 6203 to (-34.9, 161.43, 97.46) mm, rotated rx 180 ry 0 rz 180 deg; joints [-126.089, -56.789, -80.177, 61.951, 66.298, -37.033]
  MoveL 6204 to (-34.9, 161.43, 97.46) mm, rotated rx 180 ry 0 rz 180 deg; joints [-126.089, -56.789, -80.177, 61.951, 66.298, -37.033]
  Call Extruder(4.52861)
  MoveL 6205 to (-35.35, 161.1, 97.46) mm, rotated rx -180 ry 0 rz 180 deg; joints [-126.067, -56.747, -80.281, 61.947, 66.341, -36.981]
  Call Extruder(5.35652)
  MoveL 6206 to (-36.39, 160.19, 97.46) mm, rotated rx 180 ry 0 rz 180 deg; joints [-126.027, -56.64, -80.544, 61.921, 66.437, -36.845]
  Call Extruder(6.18445)
  MoveL 6207 to (-37.3, 159.15, 97.46) mm, rotated rx 180 ry 0 rz -180 deg; joints [-126.011, -56.531, -80.812, 61.875, 66.522, -36.698]
  Call Extruder(6.35176)
  MoveL 6208 to (-37.47, 158.93, 97.46) mm, rotated rx -180 ry 0 rz 180 deg; joints [-126.011, -56.509, -80.866, 61.862, 66.537, -36.667]
  MoveL 6209 to (-37.47, 158.93, 97.46) mm, rotated rx -180 ry 0 rz 180 deg; joints [-126.011, -56.509, -80.866, 61.862, 66.537, -36.667]
  Call Extruder(6.68519)
  MoveL 6210 to (-37.79, 158.48, 97.46) mm, rotated rx 180 ry 0 rz 180 deg; joints [-126.011, -56.465, -80.974, 61.838, 66.568, -36.605]
  MoveL 6211 to (-37.79, 158.48, 97.46) mm, rotated rx 180 ry 0 rz 180 deg; joints [-126.011, -56.465, -80.974, 61.838, 66.568, -36.605]
  Call Extruder(7.01743)
  MoveL 6212 to (-38.12, 158.03, 97.46) mm, rotated rx 180 ry 0 rz 180 deg; joints [-126.011, -56.421, -81.083, 61.813, 66.598, -36.544]
  MoveL 6213 to (-38.12, 158.03, 97.46) mm, rotated rx 180 ry 0 rz 180 deg; joints [-126.011, -56.421, -81.083, 61.813, 66.598, -36.544]
  Call Extruder(7.13511)
  MoveL 6214 to (-38.22, 157.85, 97.46) mm, rotated rx 180 ry 0 rz 180 deg; joints [-126.013, -56.405, -81.121, 61.802, 66.607, -36.521]
  MoveL 6215 to (-38.22, 157.85, 97.46) mm, rotated rx 180 ry 0 rz 180 deg; joints [-126.013, -56.405, -81.121, 61.802, 66.607, -36.521]
  Call Extruder(7.34283)
  MoveL 6216 to (-38.4, 157.55, 97.46) mm, rotated rx 180 ry 0 rz 180 deg; joints [-126.018, -56.378, -81.188, 61.783, 66.623, -36.481]
  MoveL 6217 to (-38.4, 157.55, 97.46) mm, rotated rx 180 ry 0 rz 180 deg; joints [-126.018, -56.378, -81.188, 61.783, 66.623, -36.481]
  Call Extruder(7.54978)
  MoveL 6218 to (-38.57, 157.25, 97.46) mm, rotated rx -180 ry 0 rz 180 deg; joints [-126.023, -56.351, -81.256, 61.763, 66.64, -36.44]
  MoveL 6219 to (-38.57, 157.25, 97.46) mm, rotated rx -180 ry 0 rz 180 deg; joints [-126.023, -56.351, -81.256, 61.763, 66.64, -36.44]
  Call Extruder(7.75595)
  MoveL 6220 to (-38.75, 156.94, 97.46) mm, rotated rx 180 ry 0 rz 180 deg; joints [-126.028, -56.323, -81.323, 61.743, 66.656, -36.4]
  MoveL 6221 to (-38.75, 156.94, 97.46) mm, rotated rx 180 ry 0 rz 180 deg; joints [-126.028, -56.323, -81.323, 61.743, 66.656, -36.4]
  Call Extruder(7.93762)
  MoveL 6222 to (-38.89, 156.67, 97.46) mm, rotated rx -180 ry 0 rz -180 deg; joints [-126.034, -56.299, -81.383, 61.724, 66.669, -36.364]
  MoveL 6223 to (-38.89, 156.67, 97.46) mm, rotated rx -180 ry 0 rz -180 deg; joints [-126.034, -56.299, -81.383, 61.724, 66.669, -36.364]
  Call Extruder(8.09561)
  MoveL 6224 to (-39, 156.42, 97.46) mm, rotated rx -180 ry 0 rz 180 deg; joints [-126.042, -56.279, -81.434, 61.706, 66.678, -36.332]
  MoveL 6225 to (-39, 156.42, 97.46) mm, rotated rx -180 ry 0 rz 180 deg; joints [-126.042, -56.279, -81.434, 61.706, 66.678, -36.332]
  Call Extruder(8.25299)
  MoveL 6226 to (-39.1, 156.17, 97.46) mm, rotated rx -180 ry 0 rz 180 deg; joints [-126.05, -56.258, -81.485, 61.687, 66.688, -36.3]
  MoveL 6227 to (-39.1, 156.17, 97.46) mm, rotated rx -180 ry 0 rz 180 deg; joints [-126.05, -56.258, -81.485, 61.687, 66.688, -36.3]
  Call Extruder(8.43571)
  MoveL 6228 to (-39.22, 155.88, 97.46) mm, rotated rx 180 ry 0 rz 180 deg; joints [-126.06, -56.234, -81.544, 61.665, 66.699, -36.263]
  MoveL 6229 to (-39.22, 155.88, 97.46) mm, rotated rx 180 ry 0 rz 180 deg; joints [-126.06, -56.234, -81.544, 61.665, 66.699, -36.263]
  Call Extruder(8.61768)
  MoveL 6230 to (-39.35, 155.58, 97.46) mm, rotated rx -180 ry 0 rz 180 deg; joints [-126.07, -56.21, -81.603, 61.643, 66.71, -36.225]
  MoveL 6231 to (-39.35, 155.58, 97.46) mm, rotated rx -180 ry 0 rz 180 deg; joints [-126.07, -56.21, -81.603, 61.643, 66.71, -36.225]
  Call Extruder(8.76501)
  MoveL 6232 to (-39.44, 155.34, 97.46) mm, rotated rx -180 ry 0 rz 180 deg; joints [-126.079, -56.191, -81.651, 61.625, 66.718, -36.195]
  MoveL 6233 to (-39.44, 155.34, 97.46) mm, rotated rx -180 ry 0 rz 180 deg; joints [-126.079, -56.191, -81.651, 61.625, 66.718, -36.195]
  Call Extruder(8.87824)
  MoveL 6234 to (-39.5, 155.15, 97.46) mm, rotated rx -180 ry 0 rz 180 deg; joints [-126.087, -56.176, -81.688, 61.609, 66.724, -36.171]
  MoveL 6235 to (-39.5, 155.15, 97.46) mm, rotated rx -180 ry 0 rz 180 deg; joints [-126.087, -56.176, -81.688, 61.609, 66.724, -36.171]
  Call Extruder(8.99103)
  MoveL 6236 to (-39.56, 154.97, 97.46) mm, rotated rx -180 ry 0 rz 180 deg; joints [-126.095, -56.162, -81.724, 61.594, 66.729, -36.148]
  MoveL 6237 to (-39.56, 154.97, 97.46) mm, rotated rx -180 ry 0 rz 180 deg; joints [-126.095, -56.162, -81.724, 61.594, 66.729, -36.148]
  Call Extruder(9.10338)
  MoveL 6238 to (-39.62, 154.78, 97.46) mm, rotated rx 180 ry 0 rz 180 deg; joints [-126.103, -56.147, -81.76, 61.579, 66.735, -36.124]
  MoveL 6239 to (-39.62, 154.78, 97.46) mm, rotated rx 180 ry 0 rz 180 deg; joints [-126.103, -56.147, -81.76, 61.579, 66.735, -36.124]
  Call Extruder(9.21528)
  MoveL 6240 to (-39.68, 154.59, 97.46) mm, rotated rx 180 ry 0 rz -180 deg; joints [-126.111, -56.132, -81.796, 61.563, 66.74, -36.101]
  MoveL 6241 to (-39.68, 154.59, 97.46) mm, rotated rx 180 ry 0 rz -180 deg; joints [-126.111, -56.132, -81.796, 61.563, 66.74, -36.101]
  Call Extruder(9.33668)
  MoveL 6242 to (-39.75, 154.38, 97.46) mm, rotated rx 180 ry 0 rz 180 deg; joints [-126.12, -56.117, -81.836, 61.546, 66.746, -36.075]
  MoveL 6243 to (-39.75, 154.38, 97.46) mm, rotated rx 180 ry 0 rz 180 deg; joints [-126.12, -56.117, -81.836, 61.546, 66.746, -36.075]
  Call Extruder(9.46747)
  MoveL 6244 to (-39.82, 154.16, 97.46) mm, rotated rx 180 ry 0 rz 180 deg; joints [-126.131, -56.099, -81.878, 61.528, 66.752, -36.047]
  MoveL 6245 to (-39.82, 154.16, 97.46) mm, rotated rx 180 ry 0 rz 180 deg; joints [-126.131, -56.099, -81.878, 61.528, 66.752, -36.047]
  Call Extruder(9.59770)
  MoveL 6246 to (-39.88, 153.94, 97.46) mm, rotated rx 180 ry 0 rz 180 deg; joints [-126.141, -56.082, -81.921, 61.509, 66.758, -36.019]
  MoveL 6247 to (-39.88, 153.94, 97.46) mm, rotated rx 180 ry 0 rz 180 deg; joints [-126.141, -56.082, -81.921, 61.509, 66.758, -36.019]
  Call Extruder(9.72737)
  MoveL 6248 to (-39.95, 153.71, 97.46) mm, rotated rx 180 ry 0 rz 180 deg; joints [-126.151, -56.065, -81.963, 61.491, 66.764, -35.992]
  MoveL 6249 to (-39.95, 153.71, 97.46) mm, rotated rx 180 ry 0 rz 180 deg; joints [-126.151, -56.065, -81.963, 61.491, 66.764, -35.992]
  Call Extruder(9.85647)
  MoveL 6250 to (-40.02, 153.49, 97.46) mm, rotated rx 180 ry 0 rz -180 deg; joints [-126.161, -56.048, -82.006, 61.472, 66.77, -35.964]
  MoveL 6251 to (-40.02, 153.49, 97.46) mm, rotated rx 180 ry 0 rz -180 deg; joints [-126.161, -56.048, -82.006, 61.472, 66.77, -35.964]
  Call Extruder(9.97155)
  MoveL 6252 to (-40.06, 153.28, 97.46) mm, rotated rx 180 ry 0 rz -180 deg; joints [-126.173, -56.033, -82.042, 61.454, 66.774, -35.939]
  MoveL 6253 to (-40.06, 153.28, 97.46) mm, rotated rx 180 ry 0 rz -180 deg; joints [-126.173, -56.033, -82.042, 61.454, 66.774, -35.939]
  Call Extruder(10.08619)
  MoveL 6254 to (-40.11, 153.08, 97.46) mm, rotated rx -180 ry 0 rz -180 deg; joints [-126.184, -56.019, -82.079, 61.436, 66.778, -35.914]
  MoveL 6255 to (-40.11, 153.08, 97.46) mm, rotated rx -180 ry 0 rz -180 deg; joints [-126.184, -56.019, -82.079, 61.436, 66.778, -35.914]
  Call Extruder(10.20037)
  MoveL 6256 to (-40.15, 152.88, 97.46) mm, rotated rx -180 ry 0 rz -180 deg; joints [-126.195, -56.004, -82.116, 61.417, 66.782, -35.889]
  MoveL 6257 to (-40.15, 152.88, 97.46) mm, rotated rx -180 ry 0 rz -180 deg; joints [-126.195, -56.004, -82.116, 61.417, 66.782, -35.889]
  Call Extruder(10.31410)
  MoveL 6258 to (-40.2, 152.67, 97.46) mm, rotated rx 180 ry 0 rz 180 deg; joints [-126.206, -55.989, -82.153, 61.399, 66.786, -35.864]
  MoveL 6259 to (-40.2, 152.67, 97.46) mm, rotated rx 180 ry 0 rz 180 deg; joints [-126.206, -55.989, -82.153, 61.399, 66.786, -35.864]
  Call Extruder(10.43952)
  MoveL 6260 to (-40.24, 152.44, 97.46) mm, rotated rx 180 ry 0 rz 180 deg; joints [-126.219, -55.973, -82.193, 61.379, 66.79, -35.837]
  MoveL 6261 to (-40.24, 152.44, 97.46) mm, rotated rx 180 ry 0 rz 180 deg; joints [-126.219, -55.973, -82.193, 61.379, 66.79, -35.837]
  Call Extruder(10.57650)
  MoveL 6262 to (-40.29, 152.2, 97.46) mm, rotated rx 180 ry 0 rz -180 deg; joints [-126.233, -55.955, -82.237, 61.356, 66.795, -35.806]
  MoveL 6263 to (-40.29, 152.2, 97.46) mm, rotated rx 180 ry 0 rz -180 deg; joints [-126.233, -55.955, -82.237, 61.356, 66.795, -35.806]
  Call Extruder(10.71287)
  MoveL 6264 to (-40.34, 151.95, 97.46) mm, rotated rx 180 ry 0 rz 180 deg; joints [-126.248, -55.937, -82.281, 61.334, 66.799, -35.776]
  MoveL 6265 to (-40.34, 151.95, 97.46) mm, rotated rx 180 ry 0 rz 180 deg; joints [-126.248, -55.937, -82.281, 61.334, 66.799, -35.776]
  Call Extruder(10.84862)
  MoveL 6266 to (-40.39, 151.7, 97.46) mm, rotated rx 180 ry 0 rz 180 deg; joints [-126.262, -55.92, -82.326, 61.311, 66.803, -35.746]
  MoveL 6267 to (-40.39, 151.7, 97.46) mm, rotated rx 180 ry 0 rz 180 deg; joints [-126.262, -55.92, -82.326, 61.311, 66.803, -35.746]
  Call Extruder(10.98377)
  MoveL 6268 to (-40.44, 151.45, 97.46) mm, rotated rx 180 ry 0 rz 180 deg; joints [-126.276, -55.902, -82.37, 61.289, 66.807, -35.716]
  MoveL 6269 to (-40.44, 151.45, 97.46) mm, rotated rx 180 ry 0 rz 180 deg; joints [-126.276, -55.902, -82.37, 61.289, 66.807, -35.716]
  Call Extruder(11.11830)
  MoveL 6270 to (-40.49, 151.2, 97.46) mm, rotated rx 180 ry 0 rz 180 deg; joints [-126.291, -55.884, -82.414, 61.266, 66.812, -35.686]
  MoveL 6271 to (-40.49, 151.2, 97.46) mm, rotated rx 180 ry 0 rz 180 deg; joints [-126.291, -55.884, -82.414, 61.266, 66.812, -35.686]
  Call Extruder(11.25223)
  MoveL 6272 to (-40.54, 150.95, 97.46) mm, rotated rx 180 ry 0 rz 180 deg; joints [-126.305, -55.867, -82.458, 61.243, 66.816, -35.655]
  MoveL 6273 to (-40.54, 150.95, 97.46) mm, rotated rx 180 ry 0 rz 180 deg; joints [-126.305, -55.867, -82.458, 61.243, 66.816, -35.655]
  Call Extruder(11.40008)
  MoveL 6274 to (-40.59, 150.67, 97.46) mm, rotated rx 180 ry 0 rz 180 deg; joints [-126.322, -55.847, -82.506, 61.218, 66.82, -35.622]
  MoveL 6275 to (-40.59, 150.67, 97.46) mm, rotated rx 180 ry 0 rz 180 deg; joints [-126.322, -55.847, -82.506, 61.218, 66.82, -35.622]
  Call Extruder(11.56181)
  MoveL 6276 to (-40.64, 150.37, 97.46) mm, rotated rx 180 ry 0 rz 180 deg; joints [-126.341, -55.826, -82.559, 61.189, 66.825, -35.585]
  MoveL 6277 to (-40.64, 150.37, 97.46) mm, rotated rx 180 ry 0 rz 180 deg; joints [-126.341, -55.826, -82.559, 61.189, 66.825, -35.585]
  Call Extruder(11.72281)
  MoveL 6278 to (-40.69, 150.06, 97.46) mm, rotated rx -180 ry 0 rz 180 deg; joints [-126.36, -55.805, -82.611, 61.161, 66.829, -35.549]
  MoveL 6279 to (-40.69, 150.06, 97.46) mm, rotated rx -180 ry 0 rz 180 deg; joints [-126.36, -55.805, -82.611, 61.161, 66.829, -35.549]
  Call Extruder(11.88308)
  MoveL 6280 to (-40.74, 149.76, 97.46) mm, rotated rx 180 ry 0 rz 180 deg; joints [-126.379, -55.784, -82.664, 61.132, 66.833, -35.512]
  MoveL 6281 to (-40.74, 149.76, 97.46) mm, rotated rx 180 ry 0 rz 180 deg; joints [-126.379, -55.784, -82.664, 61.132, 66.833, -35.512]
  Call Extruder(12.04262)
  MoveL 6282 to (-40.78, 149.45, 97.46) mm, rotated rx -180 ry 0 rz 180 deg; joints [-126.398, -55.763, -82.716, 61.103, 66.837, -35.475]
  MoveL 6283 to (-40.78, 149.45, 97.46) mm, rotated rx -180 ry 0 rz 180 deg; joints [-126.398, -55.763, -82.716, 61.103, 66.837, -35.475]
  Call Extruder(12.20144)
  MoveL 6284 to (-40.83, 149.14, 97.46) mm, rotated rx 180 ry 0 rz -180 deg; joints [-126.417, -55.742, -82.769, 61.075, 66.841, -35.439]
  MoveL 6285 to (-40.83, 149.14, 97.46) mm, rotated rx 180 ry 0 rz -180 deg; joints [-126.417, -55.742, -82.769, 61.075, 66.841, -35.439]
  Call Extruder(12.38010)
  MoveL 6286 to (-40.88, 148.8, 97.46) mm, rotated rx 180 ry 0 rz 180 deg; joints [-126.439, -55.719, -82.827, 61.041, 66.845, -35.397]
  MoveL 6287 to (-40.88, 148.8, 97.46) mm, rotated rx 180 ry 0 rz 180 deg; joints [-126.439, -55.719, -82.827, 61.041, 66.845, -35.397]
  Call Extruder(12.57854)
  MoveL 6288 to (-40.92, 148.41, 97.46) mm, rotated rx -180 ry 0 rz -180 deg; joints [-126.465, -55.693, -82.892, 61.004, 66.849, -35.351]
  MoveL 6289 to (-40.92, 148.41, 97.46) mm, rotated rx -180 ry 0 rz -180 deg; joints [-126.465, -55.693, -82.892, 61.004, 66.849, -35.351]
  Call Extruder(12.77611)
  MoveL 6290 to (-40.97, 148.02, 97.46) mm, rotated rx 180 ry 0 rz 180 deg; joints [-126.491, -55.667, -82.957, 60.966, 66.853, -35.305]
  MoveL 6291 to (-40.97, 148.02, 97.46) mm, rotated rx 180 ry 0 rz 180 deg; joints [-126.491, -55.667, -82.957, 60.966, 66.853, -35.305]
  Call Extruder(12.97282)
  MoveL 6292 to (-41.02, 147.63, 97.46) mm, rotated rx 180 ry 0 rz 180 deg; joints [-126.517, -55.641, -83.021, 60.929, 66.857, -35.259]
  MoveL 6293 to (-41.02, 147.63, 97.46) mm, rotated rx 180 ry 0 rz 180 deg; joints [-126.517, -55.641, -83.021, 60.929, 66.857, -35.259]
  Call Extruder(13.16866)
  MoveL 6294 to (-41.06, 147.25, 97.46) mm, rotated rx -180 ry 0 rz -180 deg; joints [-126.543, -55.616, -83.086, 60.891, 66.86, -35.214]
  MoveL 6295 to (-41.06, 147.25, 97.46) mm, rotated rx -180 ry 0 rz -180 deg; joints [-126.543, -55.616, -83.086, 60.891, 66.86, -35.214]
  Call Extruder(13.46406)
  MoveL 6296 to (-41.11, 146.66, 97.46) mm, rotated rx 180 ry 0 rz 180 deg; joints [-126.585, -55.578, -83.181, 60.832, 66.864, -35.144]
  MoveL 6297 to (-41.11, 146.66, 97.46) mm, rotated rx 180 ry 0 rz 180 deg; joints [-126.585, -55.578, -83.181, 60.832, 66.864, -35.144]
  Call Extruder(13.75812)
  MoveL 6298 to (-41.15, 146.07, 97.46) mm, rotated rx 180 ry 0 rz 180 deg; joints [-126.628, -55.54, -83.276, 60.773, 66.868, -35.075]
  MoveL 6299 to (-41.15, 146.07, 97.46) mm, rotated rx 180 ry 0 rz 180 deg; joints [-126.628, -55.54, -83.276, 60.773, 66.868, -35.075]
  Call Extruder(14.05086)
  MoveL 6300 to (-41.2, 145.48, 97.46) mm, rotated rx 180 ry 0 rz 180 deg; joints [-126.67, -55.502, -83.372, 60.714, 66.871, -35.006]
  MoveL 6301 to (-41.2, 145.48, 97.46) mm, rotated rx 180 ry 0 rz 180 deg; joints [-126.67, -55.502, -83.372, 60.714, 66.871, -35.006]
  Call Extruder(14.62431)
  MoveL 6302 to (-41.25, 144.32, 97.46) mm, rotated rx 180 ry 0 rz 180 deg; joints [-126.759, -55.429, -83.554, 60.594, 66.874, -34.871]
  MoveL 6303 to (-41.25, 144.32, 97.46) mm, rotated rx 180 ry 0 rz 180 deg; joints [-126.759, -55.429, -83.554, 60.594, 66.874, -34.871]
  Call Extruder(15.33827)
  MoveL 6304 to (-41.29, 142.86, 97.46) mm, rotated rx 180 ry 0 rz 180 deg; joints [-126.873, -55.34, -83.779, 60.442, 66.876, -34.702]
  Call Extruder(57.40309)
  MoveL 6305 to (-41.29, 57.14, 97.46) mm, rotated rx 180 ry 0 rz 180 deg; joints [-135.148, -50.99, -95.467, 50.044, 66.938, -25.06]
  Call Extruder(57.83164)
  MoveL 6306 to (-41.27, 56.26, 97.46) mm, rotated rx 180 ry 0 rz 180 deg; joints [-135.25, -50.955, -95.571, 49.922, 66.939, -24.964]
  MoveL 6307 to (-41.27, 56.26, 97.46) mm, rotated rx 180 ry 0 rz 180 deg; joints [-135.25, -50.955, -95.571, 49.922, 66.939, -24.964]
  Call Extruder(58.11773)
  MoveL 6308 to (-41.25, 55.68, 97.46) mm, rotated rx 180 ry 0 rz 180 deg; joints [-135.318, -50.931, -95.638, 49.84, 66.938, -24.9]
  MoveL 6309 to (-41.25, 55.68, 97.46) mm, rotated rx 180 ry 0 rz 180 deg; joints [-135.318, -50.931, -95.638, 49.84, 66.938, -24.9]
  Call Extruder(58.69247)
  MoveL 6310 to (-41.2, 54.52, 97.46) mm, rotated rx 180 ry 0 rz -180 deg; joints [-135.457, -50.885, -95.773, 49.674, 66.937, -24.774]
  MoveL 6311 to (-41.2, 54.52, 97.46) mm, rotated rx 180 ry 0 rz -180 deg; joints [-135.457, -50.885, -95.773, 49.674, 66.937, -24.774]
  Call Extruder(58.98586)
  MoveL 6312 to (-41.15, 53.93, 97.46) mm, rotated rx 180 ry 0 rz -180 deg; joints [-135.53, -50.863, -95.838, 49.588, 66.934, -24.71]
  MoveL 6313 to (-41.15, 53.93, 97.46) mm, rotated rx 180 ry 0 rz -180 deg; joints [-135.53, -50.863, -95.838, 49.588, 66.934, -24.71]
  Call Extruder(59.28059)
  MoveL 6314 to (-41.11, 53.34, 97.46) mm, rotated rx 180 ry 0 rz 180 deg; joints [-135.603, -50.841, -95.903, 49.502, 66.932, -24.646]
  MoveL 6315 to (-41.11, 53.34, 97.46) mm, rotated rx 180 ry 0 rz 180 deg; joints [-135.603, -50.841, -95.903, 49.502, 66.932, -24.646]
  Call Extruder(59.57665)
  MoveL 6316 to (-41.06, 52.75, 97.46) mm, rotated rx -180 ry 0 rz 180 deg; joints [-135.676, -50.819, -95.968, 49.416, 66.929, -24.582]
  MoveL 6317 to (-41.06, 52.75, 97.46) mm, rotated rx -180 ry 0 rz 180 deg; joints [-135.676, -50.819, -95.968, 49.416, 66.929, -24.582]
  Call Extruder(59.77292)
  MoveL 6318 to (-41.02, 52.37, 97.46) mm, rotated rx 180 ry 0 rz 180 deg; joints [-135.726, -50.805, -96.009, 49.358, 66.926, -24.541]
  MoveL 6319 to (-41.02, 52.37, 97.46) mm, rotated rx 180 ry 0 rz 180 deg; joints [-135.726, -50.805, -96.009, 49.358, 66.926, -24.541]
  Call Extruder(59.97006)
  MoveL 6320 to (-40.97, 51.98, 97.46) mm, rotated rx -180 ry 0 rz 180 deg; joints [-135.776, -50.791, -96.049, 49.3, 66.922, -24.499]
  MoveL 6321 to (-40.97, 51.98, 97.46) mm, rotated rx -180 ry 0 rz 180 deg; joints [-135.776, -50.791, -96.049, 49.3, 66.922, -24.499]
  Call Extruder(60.16807)
  MoveL 6322 to (-40.92, 51.59, 97.46) mm, rotated rx 180 ry 0 rz -180 deg; joints [-135.827, -50.777, -96.09, 49.241, 66.919, -24.458]
  MoveL 6323 to (-40.92, 51.59, 97.46) mm, rotated rx 180 ry 0 rz -180 deg; joints [-135.827, -50.777, -96.09, 49.241, 66.919, -24.458]
  Call Extruder(60.36695)
  MoveL 6324 to (-40.88, 51.2, 97.46) mm, rotated rx 180 ry 0 rz 180 deg; joints [-135.877, -50.763, -96.13, 49.183, 66.916, -24.416]
  MoveL 6325 to (-40.88, 51.2, 97.46) mm, rotated rx 180 ry 0 rz 180 deg; joints [-135.877, -50.763, -96.13, 49.183, 66.916, -24.416]
  Call Extruder(60.54602)
  MoveL 6326 to (-40.83, 50.86, 97.46) mm, rotated rx -180 ry 0 rz -180 deg; joints [-135.922, -50.751, -96.166, 49.13, 66.912, -24.379]
  MoveL 6327 to (-40.83, 50.86, 97.46) mm, rotated rx -180 ry 0 rz -180 deg; joints [-135.922, -50.751, -96.166, 49.13, 66.912, -24.379]
  Call Extruder(60.70520)
  MoveL 6328 to (-40.78, 50.55, 97.46) mm, rotated rx 180 ry 0 rz 180 deg; joints [-135.964, -50.741, -96.196, 49.083, 66.908, -24.347]
  MoveL 6329 to (-40.78, 50.55, 97.46) mm, rotated rx 180 ry 0 rz 180 deg; joints [-135.964, -50.741, -96.196, 49.083, 66.908, -24.347]
  Call Extruder(60.86511)
  MoveL 6330 to (-40.73, 50.24, 97.46) mm, rotated rx 180 ry 0 rz 180 deg; joints [-136.005, -50.73, -96.227, 49.036, 66.905, -24.314]
  MoveL 6331 to (-40.73, 50.24, 97.46) mm, rotated rx 180 ry 0 rz 180 deg; joints [-136.005, -50.73, -96.227, 49.036, 66.905, -24.314]
  Call Extruder(61.02575)
  MoveL 6332 to (-40.69, 49.94, 97.46) mm, rotated rx 180 ry 0 rz -180 deg; joints [-136.046, -50.72, -96.257, 48.989, 66.901, -24.282]
  MoveL 6333 to (-40.69, 49.94, 97.46) mm, rotated rx 180 ry 0 rz -180 deg; joints [-136.046, -50.72, -96.257, 48.989, 66.901, -24.282]
  Call Extruder(61.18711)
  MoveL 6334 to (-40.64, 49.63, 97.46) mm, rotated rx 180 ry 0 rz 180 deg; joints [-136.087, -50.71, -96.287, 48.941, 66.897, -24.249]
  MoveL 6335 to (-40.64, 49.63, 97.46) mm, rotated rx 180 ry 0 rz 180 deg; joints [-136.087, -50.71, -96.287, 48.941, 66.897, -24.249]
  Call Extruder(61.34921)
  MoveL 6336 to (-40.59, 49.33, 97.46) mm, rotated rx 180 ry 0 rz -180 deg; joints [-136.128, -50.7, -96.318, 48.894, 66.893, -24.217]
  MoveL 6337 to (-40.59, 49.33, 97.46) mm, rotated rx 180 ry 0 rz -180 deg; joints [-136.128, -50.7, -96.318, 48.894, 66.893, -24.217]
  Call Extruder(61.49740)
  MoveL 6338 to (-40.54, 49.05, 97.46) mm, rotated rx -180 ry 0 rz -180 deg; joints [-136.166, -50.69, -96.344, 48.851, 66.889, -24.188]
  MoveL 6339 to (-40.54, 49.05, 97.46) mm, rotated rx -180 ry 0 rz -180 deg; joints [-136.166, -50.69, -96.344, 48.851, 66.889, -24.188]
  Call Extruder(61.63163)
  MoveL 6340 to (-40.49, 48.8, 97.46) mm, rotated rx 180 ry 0 rz -180 deg; joints [-136.201, -50.683, -96.368, 48.811, 66.885, -24.162]
  MoveL 6341 to (-40.49, 48.8, 97.46) mm, rotated rx 180 ry 0 rz -180 deg; joints [-136.201, -50.683, -96.368, 48.811, 66.885, -24.162]
  Call Extruder(61.76647)
  MoveL 6342 to (-40.44, 48.55, 97.46) mm, rotated rx -180 ry 0 rz -180 deg; joints [-136.236, -50.675, -96.391, 48.772, 66.881, -24.135]
  MoveL 6343 to (-40.44, 48.55, 97.46) mm, rotated rx -180 ry 0 rz -180 deg; joints [-136.236, -50.675, -96.391, 48.772, 66.881, -24.135]
  Call Extruder(61.90192)
  MoveL 6344 to (-40.39, 48.3, 97.46) mm, rotated rx 180 ry 0 rz -180 deg; joints [-136.271, -50.667, -96.414, 48.732, 66.877, -24.109]
  MoveL 6345 to (-40.39, 48.3, 97.46) mm, rotated rx 180 ry 0 rz -180 deg; joints [-136.271, -50.667, -96.414, 48.732, 66.877, -24.109]
  Call Extruder(62.03798)
  MoveL 6346 to (-40.34, 48.05, 97.46) mm, rotated rx 180 ry 0 rz 180 deg; joints [-136.306, -50.659, -96.438, 48.692, 66.873, -24.083]
  MoveL 6347 to (-40.34, 48.05, 97.46) mm, rotated rx 180 ry 0 rz 180 deg; joints [-136.306, -50.659, -96.438, 48.692, 66.873, -24.083]
  Call Extruder(62.17465)
  MoveL 6348 to (-40.29, 47.8, 97.46) mm, rotated rx 180 ry 0 rz 180 deg; joints [-136.341, -50.651, -96.461, 48.653, 66.869, -24.057]
  MoveL 6349 to (-40.29, 47.8, 97.46) mm, rotated rx 180 ry 0 rz 180 deg; joints [-136.341, -50.651, -96.461, 48.653, 66.869, -24.057]
  Call Extruder(62.31193)
  MoveL 6350 to (-40.24, 47.56, 97.46) mm, rotated rx 180 ry 0 rz 180 deg; joints [-136.376, -50.643, -96.484, 48.613, 66.865, -24.031]
  MoveL 6351 to (-40.24, 47.56, 97.46) mm, rotated rx 180 ry 0 rz 180 deg; joints [-136.376, -50.643, -96.484, 48.613, 66.865, -24.031]
  Call Extruder(62.43761)
  MoveL 6352 to (-40.2, 47.33, 97.46) mm, rotated rx 180 ry 0 rz 180 deg; joints [-136.408, -50.636, -96.505, 48.577, 66.861, -24.007]
  MoveL 6353 to (-40.2, 47.33, 97.46) mm, rotated rx 180 ry 0 rz 180 deg; joints [-136.408, -50.636, -96.505, 48.577, 66.861, -24.007]
  Call Extruder(62.55156)
  MoveL 6354 to (-40.15, 47.12, 97.46) mm, rotated rx 180 ry 0 rz 180 deg; joints [-136.437, -50.63, -96.523, 48.544, 66.857, -23.985]
  MoveL 6355 to (-40.15, 47.12, 97.46) mm, rotated rx 180 ry 0 rz 180 deg; joints [-136.437, -50.63, -96.523, 48.544, 66.857, -23.985]
  Call Extruder(62.66597)
  MoveL 6356 to (-40.11, 46.92, 97.46) mm, rotated rx -180 ry 0 rz 180 deg; joints [-136.466, -50.624, -96.542, 48.511, 66.853, -23.964]
  MoveL 6357 to (-40.11, 46.92, 97.46) mm, rotated rx -180 ry 0 rz 180 deg; joints [-136.466, -50.624, -96.542, 48.511, 66.853, -23.964]
  Call Extruder(62.78083)
  MoveL 6358 to (-40.06, 46.72, 97.46) mm, rotated rx 180 ry 0 rz 180 deg; joints [-136.495, -50.617, -96.56, 48.478, 66.849, -23.943]
  MoveL 6359 to (-40.06, 46.72, 97.46) mm, rotated rx 180 ry 0 rz 180 deg; joints [-136.495, -50.617, -96.56, 48.478, 66.849, -23.943]
  Call Extruder(62.89614)
  MoveL 6360 to (-40.02, 46.51, 97.46) mm, rotated rx 180 ry 0 rz 180 deg; joints [-136.525, -50.611, -96.579, 48.445, 66.846, -23.921]
  MoveL 6361 to (-40.02, 46.51, 97.46) mm, rotated rx 180 ry 0 rz 180 deg; joints [-136.525, -50.611, -96.579, 48.445, 66.846, -23.921]
  Call Extruder(63.02552)
  MoveL 6362 to (-39.95, 46.29, 97.46) mm, rotated rx -180 ry 0 rz 180 deg; joints [-136.559, -50.605, -96.597, 48.407, 66.84, -23.898]
  MoveL 6363 to (-39.95, 46.29, 97.46) mm, rotated rx -180 ry 0 rz 180 deg; joints [-136.559, -50.605, -96.597, 48.407, 66.84, -23.898]
  Call Extruder(63.15547)
  MoveL 6364 to (-39.88, 46.06, 97.46) mm, rotated rx 180 ry 0 rz -180 deg; joints [-136.593, -50.599, -96.615, 48.37, 66.834, -23.875]
  MoveL 6365 to (-39.88, 46.06, 97.46) mm, rotated rx 180 ry 0 rz -180 deg; joints [-136.593, -50.599, -96.615, 48.37, 66.834, -23.875]
  Call Extruder(63.28598)
  MoveL 6366 to (-39.81, 45.84, 97.46) mm, rotated rx 180 ry 0 rz 180 deg; joints [-136.627, -50.593, -96.632, 48.332, 66.828, -23.852]
  MoveL 6367 to (-39.81, 45.84, 97.46) mm, rotated rx 180 ry 0 rz 180 deg; joints [-136.627, -50.593, -96.632, 48.332, 66.828, -23.852]
  Call Extruder(63.41705)
  MoveL 6368 to (-39.75, 45.62, 97.46) mm, rotated rx 180 ry 0 rz 180 deg; joints [-136.661, -50.587, -96.65, 48.294, 66.822, -23.829]
  MoveL 6369 to (-39.75, 45.62, 97.46) mm, rotated rx 180 ry 0 rz 180 deg; joints [-136.661, -50.587, -96.65, 48.294, 66.822, -23.829]
  Call Extruder(63.53870)
  MoveL 6370 to (-39.68, 45.41, 97.46) mm, rotated rx 180 ry 0 rz 180 deg; joints [-136.693, -50.582, -96.666, 48.259, 66.816, -23.808]
  MoveL 6371 to (-39.68, 45.41, 97.46) mm, rotated rx 180 ry 0 rz 180 deg; joints [-136.693, -50.582, -96.666, 48.259, 66.816, -23.808]
  Call Extruder(63.65082)
  MoveL 6372 to (-39.62, 45.22, 97.46) mm, rotated rx 180 ry 0 rz -180 deg; joints [-136.722, -50.577, -96.681, 48.227, 66.811, -23.789]
  MoveL 6373 to (-39.62, 45.22, 97.46) mm, rotated rx 180 ry 0 rz -180 deg; joints [-136.722, -50.577, -96.681, 48.227, 66.811, -23.789]
  Call Extruder(63.76339)
  MoveL 6374 to (-39.56, 45.03, 97.46) mm, rotated rx 180 ry 0 rz 180 deg; joints [-136.751, -50.572, -96.695, 48.195, 66.805, -23.77]
  MoveL 6375 to (-39.56, 45.03, 97.46) mm, rotated rx 180 ry 0 rz 180 deg; joints [-136.751, -50.572, -96.695, 48.195, 66.805, -23.77]
  Call Extruder(63.87640)
  MoveL 6376 to (-39.5, 44.85, 97.46) mm, rotated rx 180 ry 0 rz -180 deg; joints [-136.781, -50.567, -96.709, 48.163, 66.8, -23.751]
  MoveL 6377 to (-39.5, 44.85, 97.46) mm, rotated rx 180 ry 0 rz -180 deg; joints [-136.781, -50.567, -96.709, 48.163, 66.8, -23.751]
  Call Extruder(63.98986)
  MoveL 6378 to (-39.44, 44.66, 97.46) mm, rotated rx -180 ry 0 rz -180 deg; joints [-136.81, -50.562, -96.724, 48.13, 66.794, -23.731]
  MoveL 6379 to (-39.44, 44.66, 97.46) mm, rotated rx -180 ry 0 rz -180 deg; joints [-136.81, -50.562, -96.724, 48.13, 66.794, -23.731]
  Call Extruder(64.13750)
  MoveL 6380 to (-39.35, 44.42, 97.46) mm, rotated rx 180 ry 0 rz 180 deg; joints [-136.849, -50.557, -96.74, 48.088, 66.786, -23.707]
  MoveL 6381 to (-39.35, 44.42, 97.46) mm, rotated rx 180 ry 0 rz 180 deg; joints [-136.849, -50.557, -96.74, 48.088, 66.786, -23.707]
  Call Extruder(64.31984)
  MoveL 6382 to (-39.23, 44.12, 97.46) mm, rotated rx 180 ry 0 rz -180 deg; joints [-136.898, -50.55, -96.759, 48.036, 66.775, -23.678]
  MoveL 6383 to (-39.23, 44.12, 97.46) mm, rotated rx 180 ry 0 rz -180 deg; joints [-136.898, -50.55, -96.759, 48.036, 66.775, -23.678]
  Call Extruder(64.50294)
  MoveL 6384 to (-39.1, 43.83, 97.46) mm, rotated rx -180 ry 0 rz 180 deg; joints [-136.946, -50.544, -96.778, 47.983, 66.764, -23.649]
  MoveL 6385 to (-39.1, 43.83, 97.46) mm, rotated rx -180 ry 0 rz 180 deg; joints [-136.946, -50.544, -96.778, 47.983, 66.764, -23.649]
  Call Extruder(64.66062)
  MoveL 6386 to (-39, 43.58, 97.46) mm, rotated rx 180 ry 0 rz -180 deg; joints [-136.988, -50.539, -96.794, 47.938, 66.754, -23.624]
  MoveL 6387 to (-39, 43.58, 97.46) mm, rotated rx 180 ry 0 rz -180 deg; joints [-136.988, -50.539, -96.794, 47.938, 66.754, -23.624]
  Call Extruder(64.81891)
  MoveL 6388 to (-38.89, 43.33, 97.46) mm, rotated rx -180 ry 0 rz 180 deg; joints [-137.029, -50.533, -96.81, 47.893, 66.744, -23.599]
  MoveL 6389 to (-38.89, 43.33, 97.46) mm, rotated rx -180 ry 0 rz 180 deg; joints [-137.029, -50.533, -96.81, 47.893, 66.744, -23.599]
  Call Extruder(65.00093)
  MoveL 6390 to (-38.75, 43.06, 97.46) mm, rotated rx 180 ry 0 rz 180 deg; joints [-137.078, -50.528, -96.824, 47.842, 66.731, -23.572]
  MoveL 6391 to (-38.75, 43.06, 97.46) mm, rotated rx 180 ry 0 rz 180 deg; joints [-137.078, -50.528, -96.824, 47.842, 66.731, -23.572]
  Call Extruder(65.20748)
  MoveL 6392 to (-38.57, 42.75, 97.46) mm, rotated rx 180 ry 0 rz -180 deg; joints [-137.135, -50.524, -96.838, 47.783, 66.715, -23.543]
  MoveL 6393 to (-38.57, 42.75, 97.46) mm, rotated rx 180 ry 0 rz -180 deg; joints [-137.135, -50.524, -96.838, 47.783, 66.715, -23.543]
  Call Extruder(65.41481)
  MoveL 6394 to (-38.4, 42.45, 97.46) mm, rotated rx 180 ry 0 rz -180 deg; joints [-137.191, -50.519, -96.851, 47.724, 66.698, -23.514]
  MoveL 6395 to (-38.4, 42.45, 97.46) mm, rotated rx 180 ry 0 rz -180 deg; joints [-137.191, -50.519, -96.851, 47.724, 66.698, -23.514]
  Call Extruder(65.62293)
  MoveL 6396 to (-38.22, 42.15, 97.46) mm, rotated rx 180 ry 0 rz 180 deg; joints [-137.247, -50.515, -96.864, 47.665, 66.682, -23.484]
  MoveL 6397 to (-38.22, 42.15, 97.46) mm, rotated rx 180 ry 0 rz 180 deg; joints [-137.247, -50.515, -96.864, 47.665, 66.682, -23.484]
  Call Extruder(65.74064)
  MoveL 6398 to (-38.12, 41.98, 97.46) mm, rotated rx 180 ry 0 rz -180 deg; joints [-137.279, -50.513, -96.871, 47.632, 66.672, -23.468]
  MoveL 6399 to (-38.12, 41.98, 97.46) mm, rotated rx 180 ry 0 rz -180 deg; joints [-137.279, -50.513, -96.871, 47.632, 66.672, -23.468]
  Call Extruder(66.07349)
  MoveL 6400 to (-37.79, 41.52, 97.46) mm, rotated rx 180 ry 0 rz 180 deg; joints [-137.37, -50.509, -96.882, 47.538, 66.641, -23.426]
  MoveL 6401 to (-37.79, 41.52, 97.46) mm, rotated rx 180 ry 0 rz 180 deg; joints [-137.37, -50.509, -96.882, 47.538, 66.641, -23.426]
  Call Extruder(66.40752)
  MoveL 6402 to (-37.47, 41.07, 97.46) mm, rotated rx 180 ry 0 rz 180 deg; joints [-137.461, -50.505, -96.893, 47.445, 66.61, -23.384]
  MoveL 6403 to (-37.47, 41.07, 97.46) mm, rotated rx 180 ry 0 rz 180 deg; joints [-137.461, -50.505, -96.893, 47.445, 66.61, -23.384]
  Call Extruder(66.57511)
  MoveL 6404 to (-37.3, 40.85, 97.46) mm, rotated rx 180 ry 0 rz 180 deg; joints [-137.506, -50.503, -96.899, 47.399, 66.594, -23.363]
  Call Extruder(67.40442)
  MoveL 6405 to (-36.39, 39.81, 97.46) mm, rotated rx -180 ry 0 rz -180 deg; joints [-137.733, -50.502, -96.903, 47.171, 66.506, -23.27]
  Call Extruder(68.03549)
  MoveL 6406 to (-35.6, 39.11, 97.46) mm, rotated rx 180 ry 0 rz 180 deg; joints [-137.904, -50.508, -96.884, 47.003, 66.43, -23.212]
  MoveL 6407 to (-35.6, 39.11, 97.46) mm, rotated rx 180 ry 0 rz 180 deg; joints [-137.904, -50.508, -96.884, 47.003, 66.43, -23.212]
  Call Extruder(68.23306)
  MoveL 6408 to (-35.35, 38.9, 97.46) mm, rotated rx 180 ry 0 rz -180 deg; joints [-137.958, -50.511, -96.876, 46.951, 66.406, -23.194]
  Call Extruder(68.56708)
  MoveL 6409 to (-34.9, 38.57, 97.46) mm, rotated rx 180 ry 0 rz 180 deg; joints [-138.048, -50.518, -96.856, 46.865, 66.361, -23.169]
  MoveL 6410 to (-34.9, 38.57, 97.46) mm, rotated rx 180 ry 0 rz 180 deg; joints [-138.048, -50.518, -96.856, 46.865, 66.361, -23.169]
  Call Extruder(68.89991)
  MoveL 6411 to (-34.45, 38.24, 97.46) mm, rotated rx -180 ry 0 rz -180 deg; joints [-138.137, -50.524, -96.837, 46.779, 66.317, -23.143]
  MoveL 6412 to (-34.45, 38.24, 97.46) mm, rotated rx -180 ry 0 rz -180 deg; joints [-138.137, -50.524, -96.837, 46.779, 66.317, -23.143]
  Call Extruder(69.07916)
  MoveL 6413 to (-34.21, 38.07, 97.46) mm, rotated rx 180 ry 0 rz 180 deg; joints [-138.185, -50.528, -96.826, 46.733, 66.293, -23.13]
  MoveL 6414 to (-34.21, 38.07, 97.46) mm, rotated rx 180 ry 0 rz 180 deg; joints [-138.185, -50.528, -96.826, 46.733, 66.293, -23.13]
  Call Extruder(69.28727)
  MoveL 6415 to (-33.9, 37.89, 97.46) mm, rotated rx 180 ry 0 rz -180 deg; joints [-138.24, -50.534, -96.807, 46.682, 66.263, -23.117]
  MoveL 6416 to (-33.9, 37.89, 97.46) mm, rotated rx 180 ry 0 rz -180 deg; joints [-138.24, -50.534, -96.807, 46.682, 66.263, -23.117]
  Call Extruder(69.49460)
  MoveL 6417 to (-33.6, 37.71, 97.46) mm, rotated rx -180 ry 0 rz 180 deg; joints [-138.295, -50.541, -96.788, 46.631, 66.233, -23.105]
  MoveL 6418 to (-33.6, 37.71, 97.46) mm, rotated rx -180 ry 0 rz 180 deg; joints [-138.295, -50.541, -96.788, 46.631, 66.233, -23.105]
  Call Extruder(69.70115)
  MoveL 6419 to (-33.29, 37.54, 97.46) mm, rotated rx 180 ry 0 rz 180 deg; joints [-138.349, -50.547, -96.769, 46.58, 66.203, -23.093]
  MoveL 6420 to (-33.29, 37.54, 97.46) mm, rotated rx 180 ry 0 rz 180 deg; joints [-138.349, -50.547, -96.769, 46.58, 66.203, -23.093]
  Call Extruder(69.90692)
  MoveL 6421 to (-32.99, 37.36, 97.46) mm, rotated rx -180 ry 0 rz 180 deg; joints [-138.404, -50.553, -96.75, 46.53, 66.173, -23.081]
  MoveL 6422 to (-32.99, 37.36, 97.46) mm, rotated rx -180 ry 0 rz 180 deg; joints [-138.404, -50.553, -96.75, 46.53, 66.173, -23.081]
  Call Extruder(70.06522)
  MoveL 6423 to (-32.74, 37.26, 97.46) mm, rotated rx 180 ry 0 rz -180 deg; joints [-138.444, -50.56, -96.731, 46.493, 66.148, -23.075]
  MoveL 6424 to (-32.74, 37.26, 97.46) mm, rotated rx 180 ry 0 rz -180 deg; joints [-138.444, -50.56, -96.731, 46.493, 66.148, -23.075]
  Call Extruder(70.22292)
  MoveL 6425 to (-32.49, 37.15, 97.46) mm, rotated rx 180 ry 0 rz 180 deg; joints [-138.484, -50.567, -96.711, 46.457, 66.124, -23.069]
  MoveL 6426 to (-32.49, 37.15, 97.46) mm, rotated rx 180 ry 0 rz 180 deg; joints [-138.484, -50.567, -96.711, 46.457, 66.124, -23.069]
  Call Extruder(70.39301)
  MoveL 6427 to (-32.22, 37.04, 97.46) mm, rotated rx 180 ry 0 rz 180 deg; joints [-138.527, -50.574, -96.689, 46.418, 66.097, -23.063]
  MoveL 6428 to (-32.22, 37.04, 97.46) mm, rotated rx 180 ry 0 rz 180 deg; joints [-138.527, -50.574, -96.689, 46.418, 66.097, -23.063]
  Call Extruder(70.57534)
  MoveL 6429 to (-31.93, 36.91, 97.46) mm, rotated rx 180 ry 0 rz 180 deg; joints [-138.574, -50.582, -96.666, 46.377, 66.068, -23.056]
  MoveL 6430 to (-31.93, 36.91, 97.46) mm, rotated rx 180 ry 0 rz 180 deg; joints [-138.574, -50.582, -96.666, 46.377, 66.068, -23.056]
  Call Extruder(70.75692)
  MoveL 6431 to (-31.64, 36.79, 97.46) mm, rotated rx 180 ry 0 rz 180 deg; joints [-138.62, -50.59, -96.642, 46.335, 66.039, -23.05]
  MoveL 6432 to (-31.64, 36.79, 97.46) mm, rotated rx 180 ry 0 rz 180 deg; joints [-138.62, -50.59, -96.642, 46.335, 66.039, -23.05]
  Call Extruder(70.87038)
  MoveL 6433 to (-31.45, 36.73, 97.46) mm, rotated rx -180 ry 0 rz 180 deg; joints [-138.648, -50.596, -96.625, 46.311, 66.02, -23.047]
  MoveL 6434 to (-31.45, 36.73, 97.46) mm, rotated rx -180 ry 0 rz 180 deg; joints [-138.648, -50.596, -96.625, 46.311, 66.02, -23.047]
  Call Extruder(70.98339)
  MoveL 6435 to (-31.26, 36.67, 97.46) mm, rotated rx 180 ry 0 rz 180 deg; joints [-138.676, -50.601, -96.608, 46.286, 66.001, -23.045]
  MoveL 6436 to (-31.26, 36.67, 97.46) mm, rotated rx 180 ry 0 rz 180 deg; joints [-138.676, -50.601, -96.608, 46.286, 66.001, -23.045]
  Call Extruder(71.09596)
  MoveL 6437 to (-31.07, 36.61, 97.46) mm, rotated rx 180 ry 0 rz -180 deg; joints [-138.704, -50.607, -96.591, 46.262, 65.983, -23.042]
  MoveL 6438 to (-31.07, 36.61, 97.46) mm, rotated rx 180 ry 0 rz -180 deg; joints [-138.704, -50.607, -96.591, 46.262, 65.983, -23.042]
  Call Extruder(71.20808)
  MoveL 6439 to (-30.88, 36.55, 97.46) mm, rotated rx 180 ry 0 rz 180 deg; joints [-138.732, -50.613, -96.573, 46.237, 65.964, -23.04]
  MoveL 6440 to (-30.88, 36.55, 97.46) mm, rotated rx 180 ry 0 rz 180 deg; joints [-138.732, -50.613, -96.573, 46.237, 65.964, -23.04]
  Call Extruder(71.31976)
  MoveL 6441 to (-30.69, 36.49, 97.46) mm, rotated rx -180 ry 0 rz 180 deg; joints [-138.759, -50.619, -96.556, 46.213, 65.945, -23.038]
  MoveL 6442 to (-30.69, 36.49, 97.46) mm, rotated rx -180 ry 0 rz 180 deg; joints [-138.759, -50.619, -96.556, 46.213, 65.945, -23.038]
  Call Extruder(71.45084)
  MoveL 6443 to (-30.47, 36.42, 97.46) mm, rotated rx 180 ry 0 rz -180 deg; joints [-138.792, -50.626, -96.535, 46.185, 65.923, -23.035]
  MoveL 6444 to (-30.47, 36.42, 97.46) mm, rotated rx 180 ry 0 rz -180 deg; joints [-138.792, -50.626, -96.535, 46.185, 65.923, -23.035]
  Call Extruder(71.58135)
  MoveL 6445 to (-30.25, 36.35, 97.46) mm, rotated rx -180 ry 0 rz 180 deg; joints [-138.824, -50.633, -96.514, 46.157, 65.9, -23.033]
  MoveL 6446 to (-30.25, 36.35, 97.46) mm, rotated rx -180 ry 0 rz 180 deg; joints [-138.824, -50.633, -96.514, 46.157, 65.9, -23.033]
  Call Extruder(71.71129)
  MoveL 6447 to (-30.02, 36.28, 97.46) mm, rotated rx 180 ry 0 rz 180 deg; joints [-138.856, -50.64, -96.493, 46.129, 65.878, -23.031]
  MoveL 6448 to (-30.02, 36.28, 97.46) mm, rotated rx 180 ry 0 rz 180 deg; joints [-138.856, -50.64, -96.493, 46.129, 65.878, -23.031]
  Call Extruder(71.84067)
  MoveL 6449 to (-29.8, 36.22, 97.46) mm, rotated rx 180 ry 0 rz -180 deg; joints [-138.889, -50.647, -96.471, 46.101, 65.856, -23.029]
  MoveL 6450 to (-29.8, 36.22, 97.46) mm, rotated rx 180 ry 0 rz -180 deg; joints [-138.889, -50.647, -96.471, 46.101, 65.856, -23.029]
  Call Extruder(71.96263)
  MoveL 6451 to (-29.59, 36.16, 97.46) mm, rotated rx -180 ry 0 rz 180 deg; joints [-138.919, -50.655, -96.45, 46.075, 65.834, -23.027]
  MoveL 6452 to (-29.59, 36.16, 97.46) mm, rotated rx -180 ry 0 rz 180 deg; joints [-138.919, -50.655, -96.45, 46.075, 65.834, -23.027]
  Call Extruder(72.07748)
  MoveL 6453 to (-29.38, 36.12, 97.46) mm, rotated rx -180 ry 0 rz 180 deg; joints [-138.946, -50.662, -96.429, 46.052, 65.814, -23.027]
  MoveL 6454 to (-29.38, 36.12, 97.46) mm, rotated rx -180 ry 0 rz 180 deg; joints [-138.946, -50.662, -96.429, 46.052, 65.814, -23.027]
  Call Extruder(72.19188)
  MoveL 6455 to (-29.18, 36.07, 97.46) mm, rotated rx 180 ry 0 rz 180 deg; joints [-138.973, -50.669, -96.408, 46.029, 65.793, -23.027]
  MoveL 6456 to (-29.18, 36.07, 97.46) mm, rotated rx 180 ry 0 rz 180 deg; joints [-138.973, -50.669, -96.408, 46.029, 65.793, -23.027]
  Call Extruder(72.30582)
  MoveL 6457 to (-28.97, 36.03, 97.46) mm, rotated rx -180 ry 0 rz -180 deg; joints [-139, -50.676, -96.386, 46.006, 65.773, -23.027]
  MoveL 6458 to (-28.97, 36.03, 97.46) mm, rotated rx -180 ry 0 rz -180 deg; joints [-139, -50.676, -96.386, 46.006, 65.773, -23.027]
  Call Extruder(72.41931)
  MoveL 6459 to (-28.77, 35.98, 97.46) mm, rotated rx 180 ry 0 rz 180 deg; joints [-139.028, -50.683, -96.365, 45.983, 65.752, -23.027]
  MoveL 6460 to (-28.77, 35.98, 97.46) mm, rotated rx 180 ry 0 rz 180 deg; joints [-139.028, -50.683, -96.365, 45.983, 65.752, -23.027]
  Call Extruder(72.55660)
  MoveL 6461 to (-28.52, 35.93, 97.46) mm, rotated rx 180 ry 0 rz -180 deg; joints [-139.06, -50.692, -96.338, 45.956, 65.727, -23.027]
  MoveL 6462 to (-28.52, 35.93, 97.46) mm, rotated rx 180 ry 0 rz -180 deg; joints [-139.06, -50.692, -96.338, 45.956, 65.727, -23.027]
  Call Extruder(72.69327)
  MoveL 6463 to (-28.27, 35.88, 97.46) mm, rotated rx 180 ry 0 rz 180 deg; joints [-139.093, -50.702, -96.312, 45.929, 65.702, -23.027]
  MoveL 6464 to (-28.27, 35.88, 97.46) mm, rotated rx 180 ry 0 rz 180 deg; joints [-139.093, -50.702, -96.312, 45.929, 65.702, -23.027]
  Call Extruder(72.82933)
  MoveL 6465 to (-28.02, 35.83, 97.46) mm, rotated rx 180 ry 0 rz -180 deg; joints [-139.126, -50.711, -96.285, 45.902, 65.677, -23.028]
  MoveL 6466 to (-28.02, 35.83, 97.46) mm, rotated rx 180 ry 0 rz -180 deg; joints [-139.126, -50.711, -96.285, 45.902, 65.677, -23.028]
  Call Extruder(72.96478)
  MoveL 6467 to (-27.77, 35.78, 97.46) mm, rotated rx 180 ry 0 rz 180 deg; joints [-139.158, -50.72, -96.258, 45.874, 65.652, -23.028]
  MoveL 6468 to (-27.77, 35.78, 97.46) mm, rotated rx 180 ry 0 rz 180 deg; joints [-139.158, -50.72, -96.258, 45.874, 65.652, -23.028]
  Call Extruder(73.09962)
  MoveL 6469 to (-27.52, 35.73, 97.46) mm, rotated rx -180 ry 0 rz -180 deg; joints [-139.191, -50.729, -96.232, 45.847, 65.627, -23.028]
  MoveL 6470 to (-27.52, 35.73, 97.46) mm, rotated rx -180 ry 0 rz -180 deg; joints [-139.191, -50.729, -96.232, 45.847, 65.627, -23.028]
  Call Extruder(73.23385)
  MoveL 6471 to (-27.27, 35.68, 97.46) mm, rotated rx 180 ry 0 rz 180 deg; joints [-139.223, -50.738, -96.205, 45.82, 65.602, -23.029]
  MoveL 6472 to (-27.27, 35.68, 97.46) mm, rotated rx 180 ry 0 rz 180 deg; joints [-139.223, -50.738, -96.205, 45.82, 65.602, -23.029]
  Call Extruder(73.36747)
  MoveL 6473 to (-27.03, 35.63, 97.46) mm, rotated rx -180 ry 0 rz 180 deg; joints [-139.256, -50.747, -96.178, 45.793, 65.577, -23.029]
  MoveL 6474 to (-27.03, 35.63, 97.46) mm, rotated rx -180 ry 0 rz 180 deg; joints [-139.256, -50.747, -96.178, 45.793, 65.577, -23.029]
  Call Extruder(73.52957)
  MoveL 6475 to (-26.72, 35.59, 97.46) mm, rotated rx -180 ry 0 rz 180 deg; joints [-139.294, -50.758, -96.144, 45.762, 65.547, -23.031]
  MoveL 6476 to (-26.72, 35.59, 97.46) mm, rotated rx -180 ry 0 rz 180 deg; joints [-139.294, -50.758, -96.144, 45.762, 65.547, -23.031]
  Call Extruder(73.69094)
  MoveL 6477 to (-26.41, 35.54, 97.46) mm, rotated rx 180 ry 0 rz 180 deg; joints [-139.332, -50.77, -96.11, 45.73, 65.516, -23.033]
  MoveL 6478 to (-26.41, 35.54, 97.46) mm, rotated rx 180 ry 0 rz 180 deg; joints [-139.332, -50.77, -96.11, 45.73, 65.516, -23.033]
  Call Extruder(73.85158)
  MoveL 6479 to (-26.11, 35.49, 97.46) mm, rotated rx 180 ry 0 rz -180 deg; joints [-139.371, -50.782, -96.075, 45.699, 65.485, -23.034]
  MoveL 6480 to (-26.11, 35.49, 97.46) mm, rotated rx 180 ry 0 rz -180 deg; joints [-139.371, -50.782, -96.075, 45.699, 65.485, -23.034]
  Call Extruder(74.01150)
  MoveL 6481 to (-25.8, 35.44, 97.46) mm, rotated rx 180 ry 0 rz 180 deg; joints [-139.409, -50.793, -96.041, 45.668, 65.454, -23.036]
  MoveL 6482 to (-25.8, 35.44, 97.46) mm, rotated rx 180 ry 0 rz 180 deg; joints [-139.409, -50.793, -96.041, 45.668, 65.454, -23.036]
  Call Extruder(74.17068)
  MoveL 6483 to (-25.5, 35.39, 97.46) mm, rotated rx 180 ry 0 rz 180 deg; joints [-139.447, -50.805, -96.007, 45.637, 65.424, -23.038]
  MoveL 6484 to (-25.5, 35.39, 97.46) mm, rotated rx 180 ry 0 rz 180 deg; joints [-139.447, -50.805, -96.007, 45.637, 65.424, -23.038]
  Call Extruder(74.32914)
  MoveL 6485 to (-25.19, 35.34, 97.46) mm, rotated rx 180 ry 0 rz 180 deg; joints [-139.485, -50.817, -95.972, 45.606, 65.393, -23.04]
  MoveL 6486 to (-25.19, 35.34, 97.46) mm, rotated rx 180 ry 0 rz 180 deg; joints [-139.485, -50.817, -95.972, 45.606, 65.393, -23.04]
  Call Extruder(74.52802)
  MoveL 6487 to (-24.8, 35.3, 97.46) mm, rotated rx 180 ry 0 rz -180 deg; joints [-139.531, -50.832, -95.927, 45.569, 65.354, -23.044]
  MoveL 6488 to (-24.8, 35.3, 97.46) mm, rotated rx 180 ry 0 rz -180 deg; joints [-139.531, -50.832, -95.927, 45.569, 65.354, -23.044]
  Call Extruder(74.72603)
  MoveL 6489 to (-24.42, 35.25, 97.46) mm, rotated rx 180 ry 0 rz 180 deg; joints [-139.577, -50.848, -95.881, 45.531, 65.315, -23.048]
  MoveL 6490 to (-24.42, 35.25, 97.46) mm, rotated rx 180 ry 0 rz 180 deg; joints [-139.577, -50.848, -95.881, 45.531, 65.315, -23.048]
  Call Extruder(74.92317)
  MoveL 6491 to (-24.03, 35.21, 97.46) mm, rotated rx 180 ry 0 rz 180 deg; joints [-139.624, -50.864, -95.836, 45.495, 65.276, -23.052]
  MoveL 6492 to (-24.03, 35.21, 97.46) mm, rotated rx 180 ry 0 rz 180 deg; joints [-139.624, -50.864, -95.836, 45.495, 65.276, -23.052]
  Call Extruder(75.11944)
  MoveL 6493 to (-23.64, 35.16, 97.46) mm, rotated rx -180 ry 0 rz 180 deg; joints [-139.67, -50.879, -95.79, 45.458, 65.237, -23.056]
  MoveL 6494 to (-23.64, 35.16, 97.46) mm, rotated rx -180 ry 0 rz 180 deg; joints [-139.67, -50.879, -95.79, 45.458, 65.237, -23.056]
  Call Extruder(75.36513)
  MoveL 6495 to (-23.15, 35.11, 97.46) mm, rotated rx 180 ry 0 rz -180 deg; joints [-139.726, -50.899, -95.732, 45.413, 65.187, -23.062]
  MoveL 6496 to (-23.15, 35.11, 97.46) mm, rotated rx 180 ry 0 rz -180 deg; joints [-139.726, -50.899, -95.732, 45.413, 65.187, -23.062]
  Call Extruder(75.65986)
  MoveL 6497 to (-22.56, 35.07, 97.46) mm, rotated rx 180 ry 0 rz -180 deg; joints [-139.793, -50.924, -95.66, 45.361, 65.128, -23.071]
  MoveL 6498 to (-22.56, 35.07, 97.46) mm, rotated rx 180 ry 0 rz -180 deg; joints [-139.793, -50.924, -95.66, 45.361, 65.128, -23.071]
  Call Extruder(75.95325)
  MoveL 6499 to (-21.97, 35.02, 97.46) mm, rotated rx -180 ry 0 rz 180 deg; joints [-139.86, -50.949, -95.587, 45.309, 65.068, -23.079]
  MoveL 6500 to (-21.97, 35.02, 97.46) mm, rotated rx -180 ry 0 rz 180 deg; joints [-139.86, -50.949, -95.587, 45.309, 65.068, -23.079]
  Call Extruder(76.38658)
  MoveL 6501 to (-21.1, 34.97, 97.46) mm, rotated rx 180 ry 0 rz 180 deg; joints [-139.956, -50.987, -95.477, 45.235, 64.98, -23.095]
  MoveL 6502 to (-21.1, 34.97, 97.46) mm, rotated rx 180 ry 0 rz 180 deg; joints [-139.956, -50.987, -95.477, 45.235, 64.98, -23.095]
  Call Extruder(76.95874)
  MoveL 6503 to (-19.94, 34.93, 97.46) mm, rotated rx -180 ry 0 rz 180 deg; joints [-140.081, -51.038, -95.329, 45.14, 64.862, -23.117]
  MoveL 6504 to (-19.94, 34.93, 97.46) mm, rotated rx -180 ry 0 rz 180 deg; joints [-140.081, -51.038, -95.329, 45.14, 64.862, -23.117]
  Call Extruder(77.38658)
  MoveL 6505 to (-19.06, 34.91, 97.46) mm, rotated rx 180 ry 0 rz 180 deg; joints [-140.173, -51.077, -95.215, 45.072, 64.774, -23.135]
  Call Extruder(194.03526)
  MoveL 6506 to (219.06, 34.91, 97.46) mm, rotated rx 180 ry 0 rz 180 deg; joints [-155.896, -68.842, -52.837, 40.429, 39.031, -33.496]
  MoveL 6507 to (219.06, 34.91, 97.46) mm, rotated rx 180 ry 0 rz 180 deg; joints [-155.896, -68.842, -52.837, 40.429, 39.031, -33.496]
  Call Extruder(194.75084)
  MoveL 6508 to (220.52, 34.95, 97.46) mm, rotated rx 180 ry 0 rz 180 deg; joints [-155.953, -69.009, -52.479, 40.507, 38.854, -33.635]
  MoveL 6509 to (220.52, 34.95, 97.46) mm, rotated rx 180 ry 0 rz 180 deg; joints [-155.953, -69.009, -52.479, 40.507, 38.854, -33.635]
  Call Extruder(195.32557)
  MoveL 6510 to (221.68, 35, 97.46) mm, rotated rx 180 ry 0 rz -180 deg; joints [-155.997, -69.144, -52.19, 40.573, 38.713, -33.749]
  MoveL 6511 to (221.68, 35, 97.46) mm, rotated rx 180 ry 0 rz -180 deg; joints [-155.997, -69.144, -52.19, 40.573, 38.713, -33.749]
  Call Extruder(195.61897)
  MoveL 6512 to (222.27, 35.04, 97.46) mm, rotated rx 180 ry 0 rz 180 deg; joints [-156.017, -69.214, -52.04, 40.612, 38.642, -33.811]
  MoveL 6513 to (222.27, 35.04, 97.46) mm, rotated rx 180 ry 0 rz 180 deg; joints [-156.017, -69.214, -52.04, 40.612, 38.642, -33.811]
  Call Extruder(195.91369)
  MoveL 6514 to (222.86, 35.09, 97.46) mm, rotated rx -180 ry 0 rz -180 deg; joints [-156.037, -69.284, -51.891, 40.65, 38.57, -33.874]
  MoveL 6515 to (222.86, 35.09, 97.46) mm, rotated rx -180 ry 0 rz -180 deg; joints [-156.037, -69.284, -51.891, 40.65, 38.57, -33.874]
  Call Extruder(196.20975)
  MoveL 6516 to (223.45, 35.14, 97.46) mm, rotated rx 180 ry 0 rz 180 deg; joints [-156.057, -69.354, -51.74, 40.689, 38.498, -33.937]
  MoveL 6517 to (223.45, 35.14, 97.46) mm, rotated rx 180 ry 0 rz 180 deg; joints [-156.057, -69.354, -51.74, 40.689, 38.498, -33.937]
  Call Extruder(196.40603)
  MoveL 6518 to (223.84, 35.18, 97.46) mm, rotated rx 180 ry 0 rz 180 deg; joints [-156.068, -69.401, -51.64, 40.717, 38.451, -33.981]
  MoveL 6519 to (223.84, 35.18, 97.46) mm, rotated rx 180 ry 0 rz 180 deg; joints [-156.068, -69.401, -51.64, 40.717, 38.451, -33.981]
  Call Extruder(196.60317)
  MoveL 6520 to (224.22, 35.23, 97.46) mm, rotated rx -180 ry 0 rz 180 deg; joints [-156.08, -69.448, -51.539, 40.746, 38.404, -34.025]
  MoveL 6521 to (224.22, 35.23, 97.46) mm, rotated rx -180 ry 0 rz 180 deg; joints [-156.08, -69.448, -51.539, 40.746, 38.404, -34.025]
  Call Extruder(196.80118)
  MoveL 6522 to (224.61, 35.27, 97.46) mm, rotated rx -180 ry 0 rz 180 deg; joints [-156.092, -69.496, -51.438, 40.775, 38.357, -34.069]
  MoveL 6523 to (224.61, 35.27, 97.46) mm, rotated rx -180 ry 0 rz 180 deg; joints [-156.092, -69.496, -51.438, 40.775, 38.357, -34.069]
  Call Extruder(197.00005)
  MoveL 6524 to (225, 35.32, 97.46) mm, rotated rx 180 ry 0 rz -180 deg; joints [-156.103, -69.543, -51.337, 40.803, 38.31, -34.113]
  MoveL 6525 to (225, 35.32, 97.46) mm, rotated rx 180 ry 0 rz -180 deg; joints [-156.103, -69.543, -51.337, 40.803, 38.31, -34.113]
  Call Extruder(197.17913)
  MoveL 6526 to (225.34, 35.37, 97.46) mm, rotated rx 180 ry 0 rz -180 deg; joints [-156.113, -69.586, -51.246, 40.83, 38.268, -34.154]
  MoveL 6527 to (225.34, 35.37, 97.46) mm, rotated rx 180 ry 0 rz -180 deg; joints [-156.113, -69.586, -51.246, 40.83, 38.268, -34.154]
  Call Extruder(197.33832)
  MoveL 6528 to (225.65, 35.42, 97.46) mm, rotated rx 180 ry 0 rz 180 deg; joints [-156.121, -69.624, -51.165, 40.856, 38.23, -34.191]
  MoveL 6529 to (225.65, 35.42, 97.46) mm, rotated rx 180 ry 0 rz 180 deg; joints [-156.121, -69.624, -51.165, 40.856, 38.23, -34.191]
  Call Extruder(197.49823)
  MoveL 6530 to (225.96, 35.47, 97.46) mm, rotated rx 180 ry 0 rz 180 deg; joints [-156.129, -69.662, -51.083, 40.881, 38.193, -34.229]
  MoveL 6531 to (225.96, 35.47, 97.46) mm, rotated rx 180 ry 0 rz 180 deg; joints [-156.129, -69.662, -51.083, 40.881, 38.193, -34.229]
  Call Extruder(197.65887)
  MoveL 6532 to (226.26, 35.51, 97.46) mm, rotated rx 180 ry 0 rz 180 deg; joints [-156.137, -69.7, -51.002, 40.906, 38.156, -34.266]
  MoveL 6533 to (226.26, 35.51, 97.46) mm, rotated rx 180 ry 0 rz 180 deg; joints [-156.137, -69.7, -51.002, 40.906, 38.156, -34.266]
  Call Extruder(197.82023)
  MoveL 6534 to (226.57, 35.56, 97.46) mm, rotated rx -180 ry 0 rz 180 deg; joints [-156.145, -69.738, -50.92, 40.932, 38.119, -34.304]
  MoveL 6535 to (226.57, 35.56, 97.46) mm, rotated rx -180 ry 0 rz 180 deg; joints [-156.145, -69.738, -50.92, 40.932, 38.119, -34.304]
  Call Extruder(197.98233)
  MoveL 6536 to (226.87, 35.61, 97.46) mm, rotated rx -180 ry 0 rz 180 deg; joints [-156.153, -69.777, -50.839, 40.957, 38.082, -34.341]
  MoveL 6537 to (226.87, 35.61, 97.46) mm, rotated rx -180 ry 0 rz 180 deg; joints [-156.153, -69.777, -50.839, 40.957, 38.082, -34.341]
  Call Extruder(198.13052)
  MoveL 6538 to (227.15, 35.66, 97.46) mm, rotated rx -180 ry 0 rz -180 deg; joints [-156.16, -69.812, -50.764, 40.981, 38.048, -34.376]
  MoveL 6539 to (227.15, 35.66, 97.46) mm, rotated rx -180 ry 0 rz -180 deg; joints [-156.16, -69.812, -50.764, 40.981, 38.048, -34.376]
  Call Extruder(198.26476)
  MoveL 6540 to (227.4, 35.71, 97.46) mm, rotated rx 180 ry 0 rz 180 deg; joints [-156.165, -69.843, -50.696, 41.004, 38.018, -34.409]
  MoveL 6541 to (227.4, 35.71, 97.46) mm, rotated rx 180 ry 0 rz 180 deg; joints [-156.165, -69.843, -50.696, 41.004, 38.018, -34.409]
  Call Extruder(198.39960)
  MoveL 6542 to (227.65, 35.76, 97.46) mm, rotated rx 180 ry 0 rz 180 deg; joints [-156.171, -69.875, -50.628, 41.027, 37.987, -34.441]
  MoveL 6543 to (227.65, 35.76, 97.46) mm, rotated rx 180 ry 0 rz 180 deg; joints [-156.171, -69.875, -50.628, 41.027, 37.987, -34.441]
  Call Extruder(198.53505)
  MoveL 6544 to (227.9, 35.81, 97.46) mm, rotated rx 180 ry 0 rz 180 deg; joints [-156.176, -69.907, -50.561, 41.05, 37.957, -34.474]
  MoveL 6545 to (227.9, 35.81, 97.46) mm, rotated rx 180 ry 0 rz 180 deg; joints [-156.176, -69.907, -50.561, 41.05, 37.957, -34.474]
  Call Extruder(198.67111)
  MoveL 6546 to (228.15, 35.86, 97.46) mm, rotated rx 180 ry 0 rz 180 deg; joints [-156.182, -69.939, -50.493, 41.073, 37.927, -34.507]
  MoveL 6547 to (228.15, 35.86, 97.46) mm, rotated rx 180 ry 0 rz 180 deg; joints [-156.182, -69.939, -50.493, 41.073, 37.927, -34.507]
  Call Extruder(198.80779)
  MoveL 6548 to (228.4, 35.91, 97.46) mm, rotated rx 180 ry 0 rz 180 deg; joints [-156.187, -69.971, -50.424, 41.096, 37.896, -34.539]
  MoveL 6549 to (228.4, 35.91, 97.46) mm, rotated rx 180 ry 0 rz 180 deg; joints [-156.187, -69.971, -50.424, 41.096, 37.896, -34.539]
  Call Extruder(198.94507)
  MoveL 6550 to (228.64, 35.96, 97.46) mm, rotated rx 180 ry 0 rz 180 deg; joints [-156.193, -70.003, -50.356, 41.119, 37.866, -34.572]
  MoveL 6551 to (228.64, 35.96, 97.46) mm, rotated rx 180 ry 0 rz 180 deg; joints [-156.193, -70.003, -50.356, 41.119, 37.866, -34.572]
  Call Extruder(199.07074)
  MoveL 6552 to (228.87, 36, 97.46) mm, rotated rx 180 ry 0 rz 180 deg; joints [-156.198, -70.032, -50.294, 41.14, 37.838, -34.602]
  MoveL 6553 to (228.87, 36, 97.46) mm, rotated rx 180 ry 0 rz 180 deg; joints [-156.198, -70.032, -50.294, 41.14, 37.838, -34.602]
  Call Extruder(199.18469)
  MoveL 6554 to (229.08, 36.05, 97.46) mm, rotated rx 180 ry 0 rz 180 deg; joints [-156.202, -70.059, -50.237, 41.16, 37.813, -34.63]
  MoveL 6555 to (229.08, 36.05, 97.46) mm, rotated rx 180 ry 0 rz 180 deg; joints [-156.202, -70.059, -50.237, 41.16, 37.813, -34.63]
  Call Extruder(199.29908)
  MoveL 6556 to (229.28, 36.09, 97.46) mm, rotated rx 180 ry 0 rz -180 deg; joints [-156.206, -70.085, -50.181, 41.18, 37.788, -34.658]
  MoveL 6557 to (229.28, 36.09, 97.46) mm, rotated rx 180 ry 0 rz -180 deg; joints [-156.206, -70.085, -50.181, 41.18, 37.788, -34.658]
  Call Extruder(199.41393)
  MoveL 6558 to (229.48, 36.14, 97.46) mm, rotated rx 180 ry 0 rz 180 deg; joints [-156.21, -70.112, -50.125, 41.2, 37.764, -34.686]
  MoveL 6559 to (229.48, 36.14, 97.46) mm, rotated rx 180 ry 0 rz 180 deg; joints [-156.21, -70.112, -50.125, 41.2, 37.764, -34.686]
  Call Extruder(199.52924)
  MoveL 6560 to (229.69, 36.18, 97.46) mm, rotated rx -180 ry 0 rz -180 deg; joints [-156.214, -70.139, -50.068, 41.22, 37.739, -34.714]
  MoveL 6561 to (229.69, 36.18, 97.46) mm, rotated rx -180 ry 0 rz -180 deg; joints [-156.214, -70.139, -50.068, 41.22, 37.739, -34.714]
  Call Extruder(199.65360)
  MoveL 6562 to (229.9, 36.25, 97.46) mm, rotated rx 180 ry 0 rz 180 deg; joints [-156.217, -70.168, -50.006, 41.244, 37.712, -34.746]
  MoveL 6563 to (229.9, 36.25, 97.46) mm, rotated rx 180 ry 0 rz 180 deg; joints [-156.217, -70.168, -50.006, 41.244, 37.712, -34.746]
  Call Extruder(199.77848)
  MoveL 6564 to (230.12, 36.31, 97.46) mm, rotated rx 180 ry 0 rz 180 deg; joints [-156.22, -70.197, -49.945, 41.268, 37.686, -34.778]
  MoveL 6565 to (230.12, 36.31, 97.46) mm, rotated rx 180 ry 0 rz 180 deg; joints [-156.22, -70.197, -49.945, 41.268, 37.686, -34.778]
  Call Extruder(199.90388)
  MoveL 6566 to (230.33, 36.38, 97.46) mm, rotated rx -180 ry 0 rz 180 deg; joints [-156.223, -70.226, -49.883, 41.292, 37.66, -34.81]
  MoveL 6567 to (230.33, 36.38, 97.46) mm, rotated rx -180 ry 0 rz 180 deg; joints [-156.223, -70.226, -49.883, 41.292, 37.66, -34.81]
  Call Extruder(200.02979)
  MoveL 6568 to (230.55, 36.44, 97.46) mm, rotated rx 180 ry 0 rz -180 deg; joints [-156.225, -70.255, -49.821, 41.316, 37.634, -34.843]
  MoveL 6569 to (230.55, 36.44, 97.46) mm, rotated rx 180 ry 0 rz -180 deg; joints [-156.225, -70.255, -49.821, 41.316, 37.634, -34.843]
  Call Extruder(200.11575)
  MoveL 6570 to (230.69, 36.49, 97.46) mm, rotated rx 180 ry 0 rz 180 deg; joints [-156.227, -70.275, -49.779, 41.333, 37.616, -34.865]
  MoveL 6571 to (230.69, 36.49, 97.46) mm, rotated rx 180 ry 0 rz 180 deg; joints [-156.227, -70.275, -49.779, 41.333, 37.616, -34.865]
  Call Extruder(200.22765)
  MoveL 6572 to (230.88, 36.55, 97.46) mm, rotated rx -180 ry 0 rz 180 deg; joints [-156.229, -70.3, -49.724, 41.355, 37.594, -34.894]
  MoveL 6573 to (230.88, 36.55, 97.46) mm, rotated rx -180 ry 0 rz 180 deg; joints [-156.229, -70.3, -49.724, 41.355, 37.594, -34.894]
  Call Extruder(200.33999)
  MoveL 6574 to (231.07, 36.61, 97.46) mm, rotated rx 180 ry 0 rz 180 deg; joints [-156.231, -70.326, -49.67, 41.378, 37.571, -34.924]
  MoveL 6575 to (231.07, 36.61, 97.46) mm, rotated rx 180 ry 0 rz 180 deg; joints [-156.231, -70.326, -49.67, 41.378, 37.571, -34.924]
  Call Extruder(200.45278)
  MoveL 6576 to (231.26, 36.67, 97.46) mm, rotated rx -180 ry 0 rz 180 deg; joints [-156.233, -70.352, -49.615, 41.4, 37.548, -34.953]
  MoveL 6577 to (231.26, 36.67, 97.46) mm, rotated rx -180 ry 0 rz 180 deg; joints [-156.233, -70.352, -49.615, 41.4, 37.548, -34.953]
  Call Extruder(200.56601)
  MoveL 6578 to (231.45, 36.73, 97.46) mm, rotated rx -180 ry 0 rz 180 deg; joints [-156.235, -70.378, -49.56, 41.422, 37.525, -34.982]
  MoveL 6579 to (231.45, 36.73, 97.46) mm, rotated rx -180 ry 0 rz 180 deg; joints [-156.235, -70.378, -49.56, 41.422, 37.525, -34.982]
  Call Extruder(200.67969)
  MoveL 6580 to (231.64, 36.79, 97.46) mm, rotated rx -180 ry 0 rz 180 deg; joints [-156.237, -70.404, -49.505, 41.445, 37.502, -35.012]
  MoveL 6581 to (231.64, 36.79, 97.46) mm, rotated rx -180 ry 0 rz 180 deg; joints [-156.237, -70.404, -49.505, 41.445, 37.502, -35.012]
  Call Extruder(200.86165)
  MoveL 6582 to (231.93, 36.91, 97.46) mm, rotated rx -180 ry 0 rz 180 deg; joints [-156.238, -70.445, -49.417, 41.484, 37.467, -35.062]
  MoveL 6583 to (231.93, 36.91, 97.46) mm, rotated rx -180 ry 0 rz 180 deg; joints [-156.238, -70.445, -49.417, 41.484, 37.467, -35.062]
  Call Extruder(201.04437)
  MoveL 6584 to (232.22, 37.03, 97.46) mm, rotated rx 180 ry 0 rz 180 deg; joints [-156.238, -70.487, -49.329, 41.523, 37.431, -35.112]
  MoveL 6585 to (232.22, 37.03, 97.46) mm, rotated rx 180 ry 0 rz 180 deg; joints [-156.238, -70.487, -49.329, 41.523, 37.431, -35.112]
  Call Extruder(201.21479)
  MoveL 6586 to (232.49, 37.15, 97.46) mm, rotated rx -180 ry 0 rz -180 deg; joints [-156.239, -70.525, -49.247, 41.56, 37.399, -35.159]
  MoveL 6587 to (232.49, 37.15, 97.46) mm, rotated rx -180 ry 0 rz -180 deg; joints [-156.239, -70.525, -49.247, 41.56, 37.399, -35.159]
  Call Extruder(201.37278)
  MoveL 6588 to (232.74, 37.26, 97.46) mm, rotated rx -180 ry 0 rz 180 deg; joints [-156.239, -70.561, -49.171, 41.595, 37.369, -35.202]
  MoveL 6589 to (232.74, 37.26, 97.46) mm, rotated rx -180 ry 0 rz 180 deg; joints [-156.239, -70.561, -49.171, 41.595, 37.369, -35.202]
  Call Extruder(201.53139)
  MoveL 6590 to (232.99, 37.36, 97.46) mm, rotated rx -180 ry 0 rz -180 deg; joints [-156.239, -70.597, -49.095, 41.629, 37.338, -35.246]
  MoveL 6591 to (232.99, 37.36, 97.46) mm, rotated rx -180 ry 0 rz -180 deg; joints [-156.239, -70.597, -49.095, 41.629, 37.338, -35.246]
  Call Extruder(201.73755)
  MoveL 6592 to (233.29, 37.54, 97.46) mm, rotated rx 180 ry 0 rz 180 deg; joints [-156.236, -70.643, -48.997, 41.679, 37.302, -35.306]
  MoveL 6593 to (233.29, 37.54, 97.46) mm, rotated rx 180 ry 0 rz 180 deg; joints [-156.236, -70.643, -48.997, 41.679, 37.302, -35.306]
  Call Extruder(201.94450)
  MoveL 6594 to (233.6, 37.71, 97.46) mm, rotated rx -180 ry 0 rz 180 deg; joints [-156.232, -70.689, -48.899, 41.73, 37.266, -35.367]
  MoveL 6595 to (233.6, 37.71, 97.46) mm, rotated rx -180 ry 0 rz 180 deg; joints [-156.232, -70.689, -48.899, 41.73, 37.266, -35.367]
  Call Extruder(202.15222)
  MoveL 6596 to (233.9, 37.89, 97.46) mm, rotated rx 180 ry 0 rz 180 deg; joints [-156.228, -70.735, -48.801, 41.78, 37.229, -35.428]
  MoveL 6597 to (233.9, 37.89, 97.46) mm, rotated rx 180 ry 0 rz 180 deg; joints [-156.228, -70.735, -48.801, 41.78, 37.229, -35.428]
  Call Extruder(202.36072)
  MoveL 6598 to (234.21, 38.06, 97.46) mm, rotated rx 180 ry 0 rz 180 deg; joints [-156.224, -70.782, -48.703, 41.831, 37.193, -35.49]
  MoveL 6599 to (234.21, 38.06, 97.46) mm, rotated rx 180 ry 0 rz 180 deg; joints [-156.224, -70.782, -48.703, 41.831, 37.193, -35.49]
  Call Extruder(202.54027)
  MoveL 6600 to (234.45, 38.24, 97.46) mm, rotated rx 180 ry 0 rz 180 deg; joints [-156.218, -70.821, -48.62, 41.878, 37.163, -35.545]
  MoveL 6601 to (234.45, 38.24, 97.46) mm, rotated rx 180 ry 0 rz 180 deg; joints [-156.218, -70.821, -48.62, 41.878, 37.163, -35.545]
  Call Extruder(202.87368)
  MoveL 6602 to (234.9, 38.57, 97.46) mm, rotated rx -180 ry 0 rz 180 deg; joints [-156.206, -70.894, -48.466, 41.965, 37.11, -35.647]
  MoveL 6603 to (234.9, 38.57, 97.46) mm, rotated rx -180 ry 0 rz 180 deg; joints [-156.206, -70.894, -48.466, 41.965, 37.11, -35.647]
  Call Extruder(203.20828)
  MoveL 6604 to (235.35, 38.9, 97.46) mm, rotated rx 180 ry 0 rz -180 deg; joints [-156.195, -70.967, -48.311, 42.053, 37.056, -35.75]
  Call Extruder(204.03623)
  MoveL 6605 to (236.39, 39.81, 97.46) mm, rotated rx 180 ry 0 rz 180 deg; joints [-156.154, -71.144, -47.937, 42.284, 36.934, -36.015]
  Call Extruder(204.86417)
  MoveL 6606 to (237.3, 40.85, 97.46) mm, rotated rx -180 ry 0 rz -180 deg; joints [-156.097, -71.314, -47.578, 42.531, 36.828, -36.288]
  Call Extruder(205.03147)
  MoveL 6607 to (237.47, 41.07, 97.46) mm, rotated rx 180 ry 0 rz 180 deg; joints [-156.083, -71.346, -47.509, 42.582, 36.809, -36.344]
  MoveL 6608 to (237.47, 41.07, 97.46) mm, rotated rx 180 ry 0 rz 180 deg; joints [-156.083, -71.346, -47.509, 42.582, 36.809, -36.344]
  Call Extruder(205.36489)
  MoveL 6609 to (237.79, 41.52, 97.46) mm, rotated rx -180 ry 0 rz 180 deg; joints [-156.055, -71.412, -47.37, 42.685, 36.772, -36.456]
  MoveL 6610 to (237.79, 41.52, 97.46) mm, rotated rx -180 ry 0 rz 180 deg; joints [-156.055, -71.412, -47.37, 42.685, 36.772, -36.456]
  Call Extruder(205.69712)
  MoveL 6611 to (238.12, 41.98, 97.46) mm, rotated rx -180 ry 0 rz -180 deg; joints [-156.028, -71.478, -47.231, 42.789, 36.734, -36.569]
  MoveL 6612 to (238.12, 41.98, 97.46) mm, rotated rx -180 ry 0 rz -180 deg; joints [-156.028, -71.478, -47.231, 42.789, 36.734, -36.569]
  Call Extruder(205.81481)
  MoveL 6613 to (238.22, 42.15, 97.46) mm, rotated rx 180 ry 0 rz -180 deg; joints [-156.016, -71.5, -47.185, 42.826, 36.724, -36.609]
  MoveL 6614 to (238.22, 42.15, 97.46) mm, rotated rx 180 ry 0 rz -180 deg; joints [-156.016, -71.5, -47.185, 42.826, 36.724, -36.609]
  Call Extruder(206.02254)
  MoveL 6615 to (238.4, 42.45, 97.46) mm, rotated rx 180 ry 0 rz 180 deg; joints [-155.996, -71.539, -47.103, 42.893, 36.704, -36.68]
  MoveL 6616 to (238.4, 42.45, 97.46) mm, rotated rx 180 ry 0 rz 180 deg; joints [-155.996, -71.539, -47.103, 42.893, 36.704, -36.68]
  Call Extruder(206.22948)
  MoveL 6617 to (238.57, 42.75, 97.46) mm, rotated rx 180 ry 0 rz 180 deg; joints [-155.976, -71.578, -47.021, 42.959, 36.685, -36.751]
  MoveL 6618 to (238.57, 42.75, 97.46) mm, rotated rx 180 ry 0 rz 180 deg; joints [-155.976, -71.578, -47.021, 42.959, 36.685, -36.751]
  Call Extruder(206.43565)
  MoveL 6619 to (238.75, 43.06, 97.46) mm, rotated rx 180 ry 0 rz 180 deg; joints [-155.956, -71.617, -46.939, 43.026, 36.665, -36.822]
  MoveL 6620 to (238.75, 43.06, 97.46) mm, rotated rx 180 ry 0 rz 180 deg; joints [-155.956, -71.617, -46.939, 43.026, 36.665, -36.822]
  Call Extruder(206.61734)
  MoveL 6621 to (238.89, 43.33, 97.46) mm, rotated rx 180 ry 0 rz 180 deg; joints [-155.937, -71.65, -46.868, 43.085, 36.65, -36.884]
  MoveL 6622 to (238.89, 43.33, 97.46) mm, rotated rx 180 ry 0 rz 180 deg; joints [-155.937, -71.65, -46.868, 43.085, 36.65, -36.884]
  Call Extruder(206.77535)
  MoveL 6623 to (239, 43.58, 97.46) mm, rotated rx -180 ry 0 rz -180 deg; joints [-155.919, -71.678, -46.811, 43.137, 36.638, -36.939]
  MoveL 6624 to (239, 43.58, 97.46) mm, rotated rx -180 ry 0 rz -180 deg; joints [-155.919, -71.678, -46.811, 43.137, 36.638, -36.939]
  Call Extruder(206.93276)
  MoveL 6625 to (239.1, 43.83, 97.46) mm, rotated rx 180 ry 0 rz -180 deg; joints [-155.901, -71.705, -46.753, 43.189, 36.627, -36.993]
  MoveL 6626 to (239.1, 43.83, 97.46) mm, rotated rx 180 ry 0 rz -180 deg; joints [-155.901, -71.705, -46.753, 43.189, 36.627, -36.993]
  Call Extruder(207.11547)
  MoveL 6627 to (239.22, 44.12, 97.46) mm, rotated rx 180 ry 0 rz 180 deg; joints [-155.879, -71.737, -46.686, 43.25, 36.614, -37.056]
  MoveL 6628 to (239.22, 44.12, 97.46) mm, rotated rx 180 ry 0 rz 180 deg; joints [-155.879, -71.737, -46.686, 43.25, 36.614, -37.056]
  Call Extruder(207.29743)
  MoveL 6629 to (239.35, 44.42, 97.46) mm, rotated rx 180 ry 0 rz -180 deg; joints [-155.858, -71.768, -46.62, 43.311, 36.602, -37.119]
  MoveL 6630 to (239.35, 44.42, 97.46) mm, rotated rx 180 ry 0 rz -180 deg; joints [-155.858, -71.768, -46.62, 43.311, 36.602, -37.119]
  Call Extruder(207.44476)
  MoveL 6631 to (239.44, 44.66, 97.46) mm, rotated rx -180 ry 0 rz -180 deg; joints [-155.84, -71.793, -46.567, 43.36, 36.592, -37.17]
  MoveL 6632 to (239.44, 44.66, 97.46) mm, rotated rx -180 ry 0 rz -180 deg; joints [-155.84, -71.793, -46.567, 43.36, 36.592, -37.17]
  Call Extruder(207.55800)
  MoveL 6633 to (239.5, 44.85, 97.46) mm, rotated rx -180 ry 0 rz 180 deg; joints [-155.826, -71.812, -46.528, 43.399, 36.586, -37.209]
  MoveL 6634 to (239.5, 44.85, 97.46) mm, rotated rx -180 ry 0 rz 180 deg; joints [-155.826, -71.812, -46.528, 43.399, 36.586, -37.209]
  Call Extruder(207.67079)
  MoveL 6635 to (239.56, 45.03, 97.46) mm, rotated rx -180 ry 0 rz -180 deg; joints [-155.811, -71.83, -46.489, 43.437, 36.58, -37.248]
  MoveL 6636 to (239.56, 45.03, 97.46) mm, rotated rx -180 ry 0 rz -180 deg; joints [-155.811, -71.83, -46.489, 43.437, 36.58, -37.248]
  Call Extruder(207.78314)
  MoveL 6637 to (239.62, 45.22, 97.46) mm, rotated rx -180 ry 0 rz -180 deg; joints [-155.797, -71.849, -46.45, 43.475, 36.574, -37.287]
  MoveL 6638 to (239.62, 45.22, 97.46) mm, rotated rx -180 ry 0 rz -180 deg; joints [-155.797, -71.849, -46.45, 43.475, 36.574, -37.287]
  Call Extruder(207.89504)
  MoveL 6639 to (239.68, 45.41, 97.46) mm, rotated rx 180 ry 0 rz 180 deg; joints [-155.783, -71.867, -46.412, 43.513, 36.568, -37.326]
  MoveL 6640 to (239.68, 45.41, 97.46) mm, rotated rx 180 ry 0 rz 180 deg; joints [-155.783, -71.867, -46.412, 43.513, 36.568, -37.326]
  Call Extruder(208.01644)
  MoveL 6641 to (239.75, 45.62, 97.46) mm, rotated rx -180 ry 0 rz 180 deg; joints [-155.767, -71.887, -46.37, 43.554, 36.561, -37.368]
  MoveL 6642 to (239.75, 45.62, 97.46) mm, rotated rx -180 ry 0 rz 180 deg; joints [-155.767, -71.887, -46.37, 43.554, 36.561, -37.368]
  Call Extruder(208.14723)
  MoveL 6643 to (239.82, 45.84, 97.46) mm, rotated rx 180 ry 0 rz 180 deg; joints [-155.75, -71.908, -46.325, 43.599, 36.555, -37.414]
  MoveL 6644 to (239.82, 45.84, 97.46) mm, rotated rx 180 ry 0 rz 180 deg; joints [-155.75, -71.908, -46.325, 43.599, 36.555, -37.414]
  Call Extruder(208.27745)
  MoveL 6645 to (239.88, 46.06, 97.46) mm, rotated rx -180 ry 0 rz 180 deg; joints [-155.733, -71.93, -46.28, 43.644, 36.548, -37.459]
  MoveL 6646 to (239.88, 46.06, 97.46) mm, rotated rx -180 ry 0 rz 180 deg; joints [-155.733, -71.93, -46.28, 43.644, 36.548, -37.459]
  Call Extruder(208.40711)
  MoveL 6647 to (239.95, 46.29, 97.46) mm, rotated rx -180 ry 0 rz 180 deg; joints [-155.715, -71.951, -46.235, 43.689, 36.542, -37.505]
  MoveL 6648 to (239.95, 46.29, 97.46) mm, rotated rx -180 ry 0 rz 180 deg; joints [-155.715, -71.951, -46.235, 43.689, 36.542, -37.505]
  Call Extruder(208.53621)
  MoveL 6649 to (240.02, 46.51, 97.46) mm, rotated rx 180 ry 0 rz 180 deg; joints [-155.698, -71.972, -46.19, 43.734, 36.535, -37.551]
  MoveL 6650 to (240.02, 46.51, 97.46) mm, rotated rx 180 ry 0 rz 180 deg; joints [-155.698, -71.972, -46.19, 43.734, 36.535, -37.551]
  Call Extruder(208.65126)
  MoveL 6651 to (240.06, 46.72, 97.46) mm, rotated rx -180 ry 0 rz -180 deg; joints [-155.682, -71.99, -46.153, 43.773, 36.531, -37.591]
  MoveL 6652 to (240.06, 46.72, 97.46) mm, rotated rx -180 ry 0 rz -180 deg; joints [-155.682, -71.99, -46.153, 43.773, 36.531, -37.591]
  Call Extruder(208.76586)
  MoveL 6653 to (240.11, 46.92, 97.46) mm, rotated rx -180 ry 0 rz 180 deg; joints [-155.665, -72.007, -46.117, 43.813, 36.527, -37.631]
  MoveL 6654 to (240.11, 46.92, 97.46) mm, rotated rx -180 ry 0 rz 180 deg; joints [-155.665, -72.007, -46.117, 43.813, 36.527, -37.631]
  Call Extruder(208.88001)
  MoveL 6655 to (240.15, 47.12, 97.46) mm, rotated rx -180 ry 0 rz 180 deg; joints [-155.649, -72.025, -46.08, 43.853, 36.523, -37.67]
  MoveL 6656 to (240.15, 47.12, 97.46) mm, rotated rx -180 ry 0 rz 180 deg; joints [-155.649, -72.025, -46.08, 43.853, 36.523, -37.67]
  Call Extruder(208.99371)
  MoveL 6657 to (240.2, 47.33, 97.46) mm, rotated rx 180 ry 0 rz 180 deg; joints [-155.633, -72.042, -46.043, 43.893, 36.52, -37.71]
  MoveL 6658 to (240.2, 47.33, 97.46) mm, rotated rx 180 ry 0 rz 180 deg; joints [-155.633, -72.042, -46.043, 43.893, 36.52, -37.71]
  Call Extruder(209.11912)
  MoveL 6659 to (240.24, 47.55, 97.46) mm, rotated rx 180 ry 0 rz 180 deg; joints [-155.614, -72.061, -46.003, 43.936, 36.516, -37.754]
